// TIA Portal project "PLC_SecreTrap_V16" (V16)

(* hardware
DEVICE "S7-1200 station_1"  S7-1200 Station
   slot 0: "Rack_0"  S7-1200 Rack  Rack  V1.0
   slot 1: "PLC_1"  CPU 1212C DC/DC/DC  6ES7 212-1AE40-0XB0  V4.4
   slot 2: "DI 16/DQ 16x24VDC_1"  6ES7 223-1BL32-0XB0  V2.0
   slot 101: "CM 1241 (RS232)_1"  6ES7 241-1AH32-0XB0  V2.2
   slot 102: "CM 1241 (RS232)_2"  6ES7 241-1AH32-0XB0  V2.2
DEVICE "GSD device_1"  GSD.Device.PN
   slot 0: "Rack"  Rack  V1.0
   slot 0: "SINAMICS-S110-CU305PN-V4.4HF"  SINAMICS S110 CU305 PN V4.4HF/SP3  6SL3 040-0JA01-0AA0  V4.40
      slot 0: "SINAMICS S110 CU305 PN V4.4HF/SP3"  SINAMICS S110 CU305 PN V4.4HF/SP3
      slot 1: "PN-IO"  PN-IO
         slot 1: "Port 1"  Port 1
         slot 2: "Port 2"  Port 2
   slot 1: "DO Servo_1"  DO Servo
      slot 0: "Module Access Point:"  Module Access Point:
   slot 2: "DO Control Unit_1"  DO Control Unit
      slot 0: "Module Access Point:"  Module Access Point:
      slot 1: "without PROFIsafe"  without PROFIsafe
   slot 2: "Standard telegram 9, PZD-10/5"  Standard telegram 9, PZD-10/5
*)

// ===== PLC "PLC_1"  CPU 1212C DC/DC/DC =====

VAR_GLOBAL   // PLC tag table "Default tag table"
   "KM_Generator1" AT %Q0.0 : Bool;   // Contactor Generator 1
   "K_FunOFF_Generator1" AT %Q0.1 : Bool;   // Relay switch OFF Fun Generator 1
   "Tag_1" AT %M1.0 : Bool;
   "Tag_2" AT %M1.1 : Bool;
   "Tag_3" AT %M1.2 : Bool;
   "ONE" AT %M0.2 : Bool;
   "CycleInterrupt_Flag" AT %M10.0 : Bool;
   "KM_Generator2" AT %Q0.2 : Bool;   // Contactor Generator 2
   "K_FunOFF_Generator2" AT %Q0.3 : Bool;   // Relay switch OFF Fun Generator 2
   "Shutter2_LimPos1" AT %I0.5 : Bool;   // Limit switch Position 1 of Shutter 2
   "Shutter2_LimPos2" AT %I0.6 : Bool;   // Limit switch Position 2 of Shutter 2
   "Reserve1_IO" AT %I0.7 : Bool;   // Reserve 1
   "Clock_Byte" AT %MB100 : Byte;
   "Clock_10Hz" AT %M100.0 : Bool;
   "Clock_5Hz" AT %M100.1 : Bool;
   "Clock_2.5Hz" AT %M100.2 : Bool;
   "Clock_2Hz" AT %M100.3 : Bool;
   "Clock_1.25Hz" AT %M100.4 : Bool;
   "Clock_1Hz" AT %M100.5 : Bool;
   "Clock_0.625Hz" AT %M100.6 : Bool;
   "Clock_0.5Hz" AT %M100.7 : Bool;
   "Tag_4" AT %M1.3 : Bool;
   "Tag_5" AT %M1.4 : Bool;
   "Tag_6" AT %M1.5 : Bool;
   "Tag_7" AT %M1.6 : Bool;
   "EMG" AT %I0.2 : Bool;   // Emergency Stop key
   "Shutter1_LimPos1" AT %I0.3 : Bool;   // Limit switch Position 1 of Shutter 1
   "Resset_M" AT %M1.7 : Bool;
   "First_Scan" AT %M0.0 : Bool;
   "ZERO" AT %M0.3 : Bool;
   "DiagnosticStageChange" AT %M0.1 : Bool;
   "IR2" AT %I0.1 : Bool;   // Infrared sensor 2
   "IR1" AT %I0.0 : Bool;   // Infrared sensor 1
   "Shutter1_LimPos2" AT %I0.4 : Bool;   // Limit switch Position 2 of Shutter 1
   "OpenDoor_Key" AT %I1.0 : Bool;   // Open Door Key
   "CloseDoor_Key" AT %I1.1 : Bool;   // Close Door Key
   "QF_KM_Generator1" AT %I1.2 : Bool;   // State Contactor & Cercuit Breaker Generator 1
   "XRAY_Generator1" AT %I1.3 : Bool;   // X-RAY Status Generator 1
   "QF_KM_Generator2" AT %I1.4 : Bool;   // State Contactor & Cercuit Breaker Generator 2
   "XRAY_Generator2" AT %I1.5 : Bool;   // X-RAY Status Generator 2
   "RDY_Detectors" AT %I1.6 : Bool;   // Detectors is Ready to exposure
   "Fun1_Door" AT %I1.7 : Bool;   // State FUN 1 in the Door
   "Fun2_Door" AT %I2.0 : Bool;   // State FUN 2 in the Door
   "isLock_Door" AT %I2.1 : Bool;   // State Lock Door
   "Reserve2_IO" AT %I2.3 : Bool;   // Reserve 2
   "isClose_Door" AT %I2.4 : Bool;   // State Close Door
   "isFault_Door" AT %I2.5 : Bool;   // Active Fault Drive Door
   "Reserve3_IO" AT %I2.6 : Bool;   // Reserve 3
   "QF_KM_Door" AT %I2.7 : Bool;   // State QF for Door Power Source
   "QF_KM_Detectors" AT %I2.2 : Bool;   // State QF for Detector Power Source
   "K_Interlock_Generators" AT %Q0.4 : Bool;   // Relay Interlock Generators
   "Reserve1_DO" AT %Q0.6 : Bool;   // Reserve1 DO
   "Reserve2_DO" AT %Q0.7 : Bool;   // Reserve2 DO
   "K_Lock_Door" AT %Q1.0 : Bool;   // Relay Lock Door
   "HL_Door_Close" AT %Q1.1 : Bool;   // HL Door is Close
   "HL_XRAY_ON" AT %Q1.2 : Bool;   // HL X-RAY ON Status
   "TRIG_Detectors" AT %Q1.3 : Bool;   // TRIGGER to Detectors for Exposure
   "K_Fun1_Door" AT %Q1.4 : Bool;   // Relay switch ON Fun 1 Door
   "K_Fun2_Door" AT %Q1.5 : Bool;   // Relay switch ON Fun 2 Door
   "KM_Drive_Door" AT %Q1.6 : Bool;   // Contactor Drive Door
   "Reserve3_DO" AT %Q1.7 : Bool;   // Reserve 3 DO
   "Reserve4" AT %Q2.0 : Bool;   // Reserve 4 DO
   "HL_EMG" AT %Q2.1 : Bool;   // HL Emergency Stop
   "K_Open_Door" AT %Q2.3 : Bool;   // Relay Open Door
   "Reserve6_DO" AT %Q2.4 : Bool;   // Reserve6 DO
   "Reserve7_DO" AT %Q2.5 : Bool;   // Reserve7 DO
   "Reserve8_DO" AT %Q2.6 : Bool;   // Reserve8 DO
   "KM_Detectors" AT %Q2.2 : Bool;   // Contactor Detectors
   "K_Reserve" AT %Q2.7 : Bool;   // Relay Reserve
   "Tag_8" AT %Q0.5 : Bool;
END_VAR

VAR_GLOBAL CONSTANT   // PLC tag table "Default tag table"
   "LOW" : UInt := 1;
   "MIDLE" : UInt := 2;
   "HIGH" : UInt := 3;
   "NO_POWER" : UInt := 0;
   "STATUS_msg_Respose_timeout" : Word := 16#0097;   // The end of a message is recognized when there is no reply within a set time after transferring data
   "STATUS_RESPONSE_LENGHT" : Word := 16#0099;
   "STATUS_msg_CHAR_timeout" : Word := 16#0096;
   "STATUS_RESET_END" : Word := 16#0103;   // Reset complited
   "SUB_STATUS_NO_ERROR" : Word := 16#0000;
   "SYSTEM" : String := 'SYS0';   // device SYSTEM
   "GENERATOR1" : String := 'GEN1';
   "GENERATOR2" : String := 'GEN2';
   "STX" : Char := '2';
   "CR" : Char := 'D';
   "hash" : Char := '#';
   "addrSYS" : UInt := 1;   // device - System
   "addrGen1" : UInt := 2;   // device - Generator 1
   "addrGen2" : UInt := 3;   // device - Generator 2
   "addrShutter1" : UInt := 4;   // device - Shutter 1
   "addrShutter2" : UInt := 5;   // device - Shutter 2
   "addrDoor" : UInt := 6;   // device - Door
   "addrDetector" : UInt := 7;   // device - Detector
   "cmdSLEV" : UInt := 1;   // command Set Level (Presset)
   "cmdSCUR" : UInt := 3;   // command Set Current Generator
   "cmdSVLT" : UInt := 4;   // command Set Voltage Generator
   "cmdGCUR" : UInt := 5;   // command Get Current Generator
   "cmdGVLT" : UInt := 6;   // command Get Voltage Generator
   "SHUTTER1" : String := 'SHT1';
   "SHUTTER2" : String := 'SHT2';
   "DOOR" : String := 'DOOR';
   "DETECTOR" : String := 'DETC';
   "SETLEVEL" : String := 'SLEV';
   "GETLEVEL" : String := 'GLEV';
   "SETCURRENT" : String := 'SCUR';
   "SETVOLTAGE" : String := 'SVLT';
   "GETCURRENT" : String := 'GCUR';
   "GETVOLTAGE" : String := 'GVLT';
   "addrNOT" : UInt := 0;   // NOT device
   "cmdNOT" : UInt := 0;   // NOT command
   "STATUS_PC_REQ_ERROR" : Word := 16#0064;   // Error Request from PC
   "STATUS_PC_REQ_VAL_ERROR" : Word := 16#0065;   // Error Request from PC, Over value
   "cmdGLEV" : UInt := 2;   // command Get Level (Presset)
   "SETMODE" : String := 'SMOD';
   "GETMODE" : String := 'GMOD';
   "cmdSMOD" : UInt := 7;   // command Set Mode Scaner
   "cmdGMOD" : UInt := 8;   // command Get Mode Scaner
   "VP_max" : Real := 200.0;   // kV
   "VP_min" : Real := 80.0;   // kV
   "CP_max" : UInt := 6000;   // uA
   "CP_min" : UInt := 200;   // uA
   "Velo_max" : UInt := 45000;   // mm/min -> 145 ms
   "Velo_min" : UInt := 8450;   // mm/min -> 800 ms
   "SETWARM" : String := 'SWAR';
   "GETWARM" : String := 'GWAR';
   "cmdSWAR" : UInt := 9;   // command Set Warm UP Generator
   "cmdGWAR" : UInt := 10;   // command Get Warm UP Generator
   "FB_STATE_NO_PROCESSING" : UInt := 0;   // FB state: No processing
   "FB_STATE_VOLTAGE_PROGRAMM" : UInt := 1;   // FB state: Set Voltage
   "FB_STATE_CURRENT_PROGRAMM" : UInt := 2;   // FB state: Set Current
   "FB_STATE_MONITOR" : UInt := 3;   // FB state: Monitor
   "FB_STATE_FAULT_CLEAR" : UInt := 4;   // FB state: Fault Clear
   "FB_STATE_REPORT_FAULT" : UInt := 5;   // FB state: Report Fault
   "FB_STATE_HV_STATUS" : UInt := 6;   // FB state: HV Status
   "FB_STATE_X_RAY_ENABLE" : UInt := 7;   // FB state: X-RAY Enable
   "FB_STATE_WD_TIMER" : UInt := 8;   // FB state: Wath DOG Timer
   "FB_STATE_COMM_PORT_ECHO" : UInt := 9;   // FB state: Comm Port Echo
   "FB_STATE_WD_ENABLE" : UInt := 10;   // FB state: Watch Dog Enable/Disable
   "FB_STATE_WD_STATUS" : UInt := 11;   // FB state: Watch Dog
   "SETXRAY" : String := 'SRAY';
   "GETXRAY" : String := 'GRAY';
   "cmdSRAY" : UInt := 12;   // command Set X-RAY
   "cmdGRAY" : UInt := 11;   // command Get X-RAY
   "STATUS_msg_timeout" : UInt := 16#0095;
   "SETCLEAR" : String := 'SCLR';
   "cmdSCLR" : UInt := 13;   // command Reset
   "cmdGFLT" : UInt := 14;   // Command Get Fault
   "GETFAULT" : String := 'GFLT';
   "stageCycleShutter" : UInt := 10;   // Cycle Test Shutter
   "stageWaitGuest" : UInt := 0;   // Stage of waiting Guest
   "stagePrepareScan" : UInt := 1;   // Stage of preparing to scan
   "stageScaning" : UInt := 2;   // Stage of Scaning
   "stageOpenDoor" : UInt := 3;   // Stage of Opening the door
   "DRIVE1" : String := 'DRV1';   // device - Drive 1
   "DRIVE2" : String := 'DRV2';   // device - Drive 2
   "SETPOSITION" : String := 'SPOS';   // Set position of shutter
   "addrServoDrive1" : UInt := 8;   // device - Drive 1
   "addrServoDrive2" : UInt := 9;   // device - Drive 2
   "cmdSPOS" : UInt := 15;   // command positioning Drive
   "modeAUTO" : UInt := 3;   // mode AUTO
   "modeJOG" : UInt := 2;   // mode JOG
   "modeLIMITED" : UInt := 1;   // mode LIMITED
   "modeOFF" : UInt := 0;   // mode OFF
   "modeSERVIСE" : UInt := 4;   // mode Service
   "CountERR" : UInt := 3;   // Error Count
   "STATUS_SUBSEQUENT_CALL" : Word := 16#0102;   // Subsequent call during active processing without further details
   "STATUS_FIRST_CALL" : Word := 16#0101;   // First call after incoming new job (rising edge 'enable')
   "STATUS_NO_CALL" : Word := 16#0100;   // No job being currently processed
   "ERR_UNDEFINED_STATE" : Word := 16#0106;   // Error: due to an undefined state in state machine
   "ERR_Response_Generator" : Word := 16#0105;   // Error: response from generator not match argument CMD
   "ERR_NO_Response_Generator" : Word := 16#0104;   // Error: response from generator not match argument CMD
   "SETRESET" : String := 'SRES';
   "cmdSRES" : UInt := 16;   // command Set Reset logics
   "SETSCAN" : String := 'SCAN';   // Set Scan
   "cmdSCAN" : UInt := 17;   // command Set Scan
   "Xexposure" : DInt := 113000;   // Distance of shuter moove
   "AccShutter" : DInt := 57600;   // mm/min2, acceleration of shutter
   "TexposureMAX" : UInt := 800;   // ms, Maximum exposure time
   "TexposureMIN" : UInt := 145;   // ms, Minimum exposure time
   "SETPRES1" : String := 'SPR1';   // Set preset 1. Exposure tim in ms
   "SETPRES2" : String := 'SPR2';   // Set preset 2. Exposure tim in ms
   "SETPRES3" : String := 'SPR3';   // Set preset 3. Exposure tim in ms
   "cmdSPRESET1" : UInt := 18;   // Set preset 1. Exposure tim in ms
   "cmdSPRESET2" : UInt := 19;   // Set preset 2. Exposure tim in ms
   "cmdSPRESET3" : UInt := 20;   // Set preset 3. Exposure tim in ms
END_VAR

TYPE "typeGeneratorDATA"
   STRUCT
      VP_Programm : Real;   // Voltage Program
      CP_Programm : UInt;   // Current Program
      VP_Monitor : Real;   // Voltage Monitor
      CP_Monitor : UInt;   // Current Monitor
      T_Monitor : Real;   // Temperature Monitor
      FIL_Monitor : UInt;   // Filament Monitor
      X_RAY_Enable : Bool;   // Enable X-RAY
      X_RAY_Status : Bool;   // Monitir X-RAY status
      WDTE : Bool;   // Watch Dog Timer
      FREV : Bool;   // Comm Port Echo
      WDOG : Bool;   // Watch Dog Timer Enable/Disable
      WDOG_Status : Bool;
      FLT : Array[0..9] of Bool;   // Report Fault
      CMD_VP : Bool;   // Command Voltage Program
      CMD_CP : Bool;   // Command Current Program
      CMD_MON : Bool;   // Command Voltage/Current/Temperature/Filament Monitor
      CMD_CLR : Bool;   // Command Fault Clear
      CMD_FLT : Bool;   // Command Report Fault
      CMD_STAT : Bool;   // Command HV Status
      CMD_ENBL : Bool;   // Command X-Ray Enable
      CMD_WDTE : Bool;   // Command Watch Dog Timer
      CMD_FREV : Bool;   // Command Comm Port Echo
      CMD_WDOG : Bool;   // Command Watch Dog Enable/Disable
      CMD_WSTAT : Bool;   // Command Watch Dog Status
      CMD_CYCLE : Bool;   // CYCLE of executing Command
      CMD_VP_Ok : Bool;
      CMD_CP_Ok : Bool;
      DiagnosticCMD : Array[0..15] of "typeDiagnostics";
      cmd_Nunmber : UInt;   // Number executed command
      cmdDone : Bool;   // Command is done
      cmdError : Bool;   // Error
      cmdState : Word;   // Command status
   END_STRUCT;
   // // FLT[0] : Regulation
   // // FLT[1] : Interlock Open
   // // FLT[2] : Cathode Over KV Fault
   // // FLT[3] : Anode Over KV Fault
   // // FLT[4] : Over Temperature Fault
   // // FLT[5] : Arc Fault
   // // FLT[6] : Over Current Fault
   // // FLT[7] : Power Limit Fault
   // // FLT[8] : Over Voltage Fault
END_TYPE

TYPE "typeDiagnostics"
TITLE = typeDiagnosticsTemplate
   STRUCT
      status : Word;   // Status of the Block or error identification when error occurred
      count : UInt;   // Count of error occurred
   END_STRUCT;
END_TYPE

TYPE "typePresset"
   STRUCT
      VP : Real;   // Voltage rogramm
      CP : UInt;   // Current rogramm
      Velocity : DInt;   // Velocity shutter
      Texposure : UInt;   // Exposure time for shutter
      Ttrigger : Time;   // Trigger time for CareRay
   END_STRUCT;
END_TYPE

TYPE "typeTEL9"
   STRUCT
      OFF1 : Bool;   // 1 = On, 0 = Off (OFF1)
      OFF2 : Bool;   // 1 = No Coast Stop, 0 = Coast Stop (OFF2)
      OFF3 : Bool;   // 1 = No Quick Stop, 0 = Quick Stop (OFF3)
      enableOperation : Bool;   // 1 = Enable operation
      rejectTraversingTask : Bool;   // 0 = Reject active traversing task
      intermediateStop : Bool;   // 0 = Intermediate STOP active traversing task
      acknowledgeError : Bool;   // Acknowledge faults (0 -> 1)
      jog1 : Bool;   // Jog 1 signal
      jog2 : Bool;   // Jog 2 signal
      startHomingProcedure : Bool;   // Start homing procedure
      activateTraversingTask : Bool;   // Activate traversing task
      traversingTaskSelection : UInt;   // Select traversing task (0..1023)
      submode : Bool;   // Submode: 0 = program 1 = Manual data input (MDI)
      stw2 : Word;   // Control word 2 (STW2)
      targetPositionMDI : DInt;   // MDI target position
      velocityMDI : DInt;   // MDI velocity
      accelerationOverrideMDI : Real;   // MDI override of acceleration [%]
      decelerationOverrideMDI : Real;   // MDI override of deceleration [%]
      positioningModeMDI : Bool;   // Positioning 0 = relative 1 = absolute
      directionPositiveMDI : Bool;   // Modulo axis: Absolute positioning in positive direction. If directionPosMDI = directionNegMDI positioning via shortest way.
      directionNegativeMDI : Bool;   // Modulo axis: Absolute positioning in negative direction. If directionNegMDI = directionPosMDI positioning via shortest way.
      operationEnabled : Bool;   // Operation enabled
      switchingOnInhibited : Bool;   // Switching on inhibited
      faultActive : Bool;   // Fault present
      warningActive : Bool;   // Warning present
      homePositionSet : Bool;   // Home position set (axis homed)
      targetPositionReached : Bool;   // Target position reached
      driveStopped : Bool;   // A traversing task has been completed or standstill for intermediate stop
      traversingTaskAcknowledged : Bool;   // A new traversing task or MDI setpoint was started
      actualPosition : DInt;   // Actual position
      activeTraversingTask : UInt;   // Active traversing task
      zsw1 : Word;   // Status word 1
      zsw2 : Word;   // Status word 2
      error : Bool;   // Error active, check status and diagId
      status : Word;   // Status output (7002 = FB in operation; 8xxx = error code)
      diagId : DWord;   // Error codes of the cyclic system function blocks GETIO / SETIO
   END_STRUCT;
END_TYPE

TYPE "typeREQ"
   STRUCT
      STX : Byte := '2';
      ADDR : Array[0..3] of Byte;
      hash1 : Byte := '#';
      CMD : Array[0..3] of Byte;
      hash2 : Byte := '#';
      VALUE : Array[0..3] of Byte;
      CR : Byte := 'D';
   END_STRUCT;
END_TYPE

TYPE "typeRESP"
   STRUCT
      STX : Byte := '2';
      ADDR : Array[0..3] of Byte;
      hash1 : Byte := '#';
      CMD : Array[0..3] of Byte;
      hash2 : Byte := '#';
      VALUE : Array[0..3] of Byte;
      CR : Byte := 'D';
   END_STRUCT;
END_TYPE

TYPE "typeWarmTable"
   STRUCT
      VP : Array[1..10] of Real;
      CP : Array[1..10] of UInt;
      T : Array[1..3] of Time;
   END_STRUCT;
END_TYPE

DATA_BLOCK "temp"   // DB2
{ S7_Optimized_Access := 'TRUE' }
VERSION : 0.1
   VAR RETAIN
      Time_Temp : Array[0..18] of DTL;
      Temperature : Array[0..18] of Real;
      index_temperature : UInt;
   END_VAR
   VAR
      "test.temperature_EN" : Bool;
      temp_XRAY_ON : Bool;
      front : Bool;
      rise1 : Bool;
      rize2 : Bool;
      cycleShutter : Bool;
      "T1_X-RAY" : DTL;
      "T2_X-RAY" : DTL;
      T_XRAY : Time;
      rise2 : Bool;
      para : UInt;
      err : Bool;
   END_VAR
BEGIN
END_DATA_BLOCK

// folder: CMD

DATA_BLOCK "PCtoPLC_DB"   // DB12
{ S7_Optimized_Access := 'TRUE' }
VERSION : 0.1
// stored: InstanceOfName ParcingCMD
"ParcingCMD"
BEGIN
END_DATA_BLOCK

DATA_BLOCK "SateMaсhineCMD_DB"   // DB15
{ S7_Optimized_Access := 'TRUE' }
VERSION : 0.1
// stored: InstanceOfName SateMaсhineCMD
"SateMaсhineCMD"
BEGIN
END_DATA_BLOCK

// folder: Drive

DATA_BLOCK "DriveStage_DB_1"   // DB7
{ S7_Optimized_Access := 'TRUE' }
VERSION : 0.1
// stored: InstanceOfName DrivesStage
"DrivesStage"
BEGIN
END_DATA_BLOCK

DATA_BLOCK "PD_TEL9_DrivePos_DB_1"   // DB17
{ S7_Optimized_Access := 'TRUE' }
AUTHOR : SIEMENS
VERSION : 0.1
// stored: InstanceOfName PD_TEL9_DrivePos
"PD_TEL9_DrivePos"
BEGIN
END_DATA_BLOCK

DATA_BLOCK "TEL9_Drive1"   // DB20
{ S7_Optimized_Access := 'TRUE' }
VERSION : 0.1
BEGIN
END_DATA_BLOCK

DATA_BLOCK "DriveStage_DB_2"   // DB41
{ S7_Optimized_Access := 'TRUE' }
VERSION : 0.1
// stored: InstanceOfName DrivesStage
"DrivesStage"
BEGIN
END_DATA_BLOCK

DATA_BLOCK "PD_TEL9_DrivePos_DB_2"   // DB42
{ S7_Optimized_Access := 'TRUE' }
AUTHOR : SIEMENS
VERSION : 0.1
// stored: InstanceOfName PD_TEL9_DrivePos
"PD_TEL9_DrivePos"
BEGIN
END_DATA_BLOCK

DATA_BLOCK "TEL9_Drive2"   // DB43
{ S7_Optimized_Access := 'TRUE' }
VERSION : 0.1
BEGIN
END_DATA_BLOCK

// folder: Generators

DATA_BLOCK "Generator1_DIO_DB"   // DB1
{ S7_Optimized_Access := 'TRUE' }
VERSION : 0.1
// stored: InstanceOfName GeneratorDIO
"GeneratorDIO"
BEGIN
   statString := '7770';
END_DATA_BLOCK

DATA_BLOCK "WarmTable"   // DB3
{ S7_Optimized_Access := 'TRUE' }
VERSION : 0.1
BEGIN
   T[1] := T#300s;
   T[2] := T#60s;
   T[3] := T#30s;
   VP[1] := 80.0;
   VP[2] := 90.0;
   VP[3] := 100.0;
   VP[4] := 110.0;
   VP[5] := 120.0;
   VP[6] := 130.0;
   VP[7] := 140.0;
   VP[8] := 150.0;
   VP[9] := 160.0;
   VP[10] := 160.0;
   CP[1] := 200;
   CP[2] := 530;
   CP[3] := 860;
   CP[4] := 1190;
   CP[5] := 1520;
   CP[6] := 1850;
   CP[7] := 2180;
   CP[8] := 2510;
   CP[9] := 2840;
   CP[10] := 3120;
END_DATA_BLOCK

DATA_BLOCK "GeneratorDATA_1"   // DB6
{ S7_Optimized_Access := 'TRUE' }
VERSION : 0.1
BEGIN
END_DATA_BLOCK

DATA_BLOCK "GenOperate1_DB"   // DB8
{ S7_Optimized_Access := 'TRUE' }
VERSION : 0.1
// stored: InstanceOfName GenOperate
"GenOperate"
BEGIN
END_DATA_BLOCK

DATA_BLOCK "GenOperate2_DB"   // DB16
{ S7_Optimized_Access := 'TRUE' }
VERSION : 0.1
// stored: InstanceOfName GenOperate
"GenOperate"
BEGIN
END_DATA_BLOCK

DATA_BLOCK "GeneratorWarm1_DB"   // DB34
{ S7_Optimized_Access := 'TRUE' }
VERSION : 0.1
// stored: InstanceOfName GeneratorWarm
"GeneratorWarm"
BEGIN
END_DATA_BLOCK

DATA_BLOCK "GeneratorDATA_2"   // DB36
{ S7_Optimized_Access := 'TRUE' }
VERSION : 0.1
BEGIN
END_DATA_BLOCK

DATA_BLOCK "GeneratorWarm2_DB"   // DB51
{ S7_Optimized_Access := 'TRUE' }
VERSION : 0.1
// stored: InstanceOfName GeneratorWarm
"GeneratorWarm"
BEGIN
END_DATA_BLOCK

DATA_BLOCK "Generator2_DIO_DB"   // DB52
{ S7_Optimized_Access := 'TRUE' }
VERSION : 0.1
// stored: InstanceOfName GeneratorDIO
"GeneratorDIO"
BEGIN
   statString := '7770';
END_DATA_BLOCK

// folder: Global_DATA

DATA_BLOCK "DIODATA"   // DB9
{ S7_Optimized_Access := 'TRUE' }
VERSION : 0.1
   VAR
      DI : Struct
         IR1_I0_0 : Bool;   // Infrared Sensor 1
         IR2_I0_1 : Bool;   // Infrared Sensor 2
         EMG_I0_2 : Bool;   // Key Emergensy Stop
         Pos1_Shutter1_I0_3 : Bool;   // Position Switch 1 of Shutter 1
         Pos2_Shutter1_I0_4 : Bool;   // Position Switch 2 of Shutter 1
         Pos1_Shutter2_I0_5 : Bool;   // Position Switch 2 of Shutter 1
         Pos2_Shutter2_I0_6 : Bool;   // Position Switch 2 of Shutter 1
         Reserve1_I0_7 : Bool;   // Reserve1
         OpenDoor_I1_0 : Bool;   // Key Open Door
         CloseDoor_I1_1 : Bool;   // Key Close Door
         QF_KM_Drive1_I1_2 : Bool;   // State Contactor & Cercuit Breaker Drive 1
         XRAY_Generator1_I1_3 : Bool;   // X-RAY Status Generator 1
         QF_KM_Drive2_I1_4 : Bool;   // State Contactor & Cercuit Breaker Drive 2
         XRAY_Generator2_I1_5 : Bool;   // X-RAY Status Generator 2
         RDY_Detectors_I1_6 : Bool;   // Detectors is Ready to exposure
         Fun1_Door_I1_7 : Bool;   // State FUN 1 in the Door
         Fun2_Door_I2_0 : Bool;   // State FUN 2 in the Door
         LockDoor_I2_1 : Bool;   // State Lock Door
         QF_KM_Detectors_I2_2 : Bool;   // State QF for Detector Power Source
         Reserve2_I2_3 : Bool;   // Reserve2
         Close_Door_I2_4 : Bool;   // State Close Door
         Fault_Door_I2_5 : Bool;   // State Fault Drive Door
         Reserve3_I2_6 : Bool;   // Reserve3
         Reserve4_I2_7 : Bool;   // Reserve4
      END_STRUCT;
      "DO" : Struct
         KM_Drive1_Q0_0 : Bool;   // Contactor Drive 1
         K_FunOFF_Generator1_Q0_1 : Bool;   // Relay switch OFF Fun Generator 1
         KM_Drive2_Q0_2 : Bool;   // Contactor Drive 2
         K_FunOFF_Generator2_Q0_3 : Bool;   // Relay switch OFF Fun Generator 2
         K_Interlock_Generators_Q0_4 : Bool;   // Relay Interlock Generators
         K_Open_Door_Q0_5 : Bool;   // Relay Open Door
         Reserve1_Q0_6 : Bool;   // Reserve 1 DO
         Reserve2_Q0_7 : Bool;   // Reserve 2 DO
         K_Lock_Door_Q1_0 : Bool;   // Relay Lock Door
         HL_Door_Close_Q1_1 : Bool;   // HL Door is Close
         HL_XRAY_ON_Q1_2 : Bool;   // HL X-RAY ON Status
         TRIG_Detectors_Q1_3 : Bool;   // TRIGGER to Detectors for Exposure
         K_Fun1_Door_Q1_4 : Bool;   // Relay switch ON Fun 1 Door
         K_Fun2_Door_Q1_5 : Bool;   // Relay switch ON Fun 2 Door
         KM_Drive_Door_Q1_6 : Bool;   // Contactor Drive Door
         Reserve3_Q1_7 : Bool;   // Reserve 3 DO
         Reserve4_Q2_0 : Bool;   // Reserve 4 DO
         HL_EMG_Q2_1 : Bool;   // HL Emergency Stop
         KM_Detectors_Q2_2 : Bool;   // Contactor Detectors
         Reserve5_Q2_3 : Bool;   // Reserve 5 DO
         Reserve6_Q2_4 : Bool;   // Reserve 6 DO
         Reserve7_Q2_5 : Bool;   // Reserve 7 DO
         Reserve8_Q2_6 : Bool;   // Reserve 8 DO
         K_Reserve_Q2_7 : Bool;   // Relay Reserve
      END_STRUCT;
   END_VAR
BEGIN
END_DATA_BLOCK

DATA_BLOCK "CmdDATA"   // DB10
{ S7_Optimized_Access := 'TRUE' }
VERSION : 0.1
   VAR
      REQ : String[16] := '               ';
      RESP : String[16] := '               ';
   END_VAR
BEGIN
END_DATA_BLOCK

DATA_BLOCK "PressetDATA"   // DB13
{ S7_Optimized_Access := 'TRUE' }
VERSION : 0.1
   VAR RETAIN
      Shutter1 : Struct
         POS1 : DInt := 5000;   // um Position Start Sgutter
         POS2 : DInt := 147000;   // um Position Stop Sgutter
      END_STRUCT;
      Shutter2 : Struct
         POS1 : DInt := 5000;   // um Position Start Sgutter
         POS2 : DInt := 147000;   // um Position Stop Sgutter
      END_STRUCT;
      GUEST : Array[0..3] of "typePresset";
   END_VAR
BEGIN
   GUEST[0].Velocity := 0;   // mm/min
   GUEST[1].Velocity := 8480;   // 8480 mm/min 800 ms
   GUEST[2].Velocity := 17000;   // 17000 mm/min 400 ms
   GUEST[3].Velocity := 45000;   // 45000 mm/min 145 ms
   GUEST[1].VP := 80.0;   // kV
   GUEST[1].CP := 200;   // uA
   GUEST[2].VP := 80.0;   // kV
   GUEST[2].CP := 200;   // uA
   GUEST[3].VP := 80.0;   // kV
   GUEST[3].CP := 200;   // uA
   GUEST[1].Texposure := 800;
   GUEST[2].Texposure := 400;
   GUEST[3].Texposure := 140;
   // GUEST[0].VP : kV
   // GUEST[0].CP : uA
END_DATA_BLOCK

DATA_BLOCK "GlobalDATA"   // DB14
{ S7_Optimized_Access := 'TRUE' }
VERSION : 0.1
   VAR
      N_Presset : UInt := 0;   // 0 - NO Scan, 1 - Low. 2 - Medium, 3 - High
      CountShot : UInt := 2;   // 1- one shot, 2- two shot
      modeDrive : Bool;   // 0-MDI 1-JOG
      readyToScan : Bool;   // 0 - is not ready to scan, 1- ready to scan
      readyData : Bool;   // 0 - Images not ready, 1 - Images ready
      modeScan : UInt := 0;   // 0 to 4. 0 - OFF, 1 - Limited, 2-JOG, 3-AUTO, 4-Service
      stageScan : UInt;   // 0 - WaitGuest, 1 - PrepareScan, 2 - Scaning, 3 - OpenDoor
      startScan : Bool;   // 0 - no Scan, 1 - Set Scan
      newPreset : Bool;   // 0 - no Preset, 1- recive new preset
      Scan_XRAY : Bool;   // 0 - Scan without XRAY, 1 - Scan with X-RAY
      cmdReset : Struct   // Resset Command
         Global : Bool;   // Reset global logic
         Drive1 : Bool;   // Reset drive 1 logic and Fault
         Drive2 : Bool;   // Reset drive 2 logic and Fault
         Generator1 : Bool;   // Reset Generator 1 logic
         Generator2 : Bool;   // Reset Generator 2 logic
         Door : Bool;   // Reset Drive door
         Detector : Bool;   // Reset Detector logic
      END_STRUCT;
      Shutter1 : Struct   // Command and state of Shutter 1
         cmdCycle : Bool;   // Command cycle moving in Service mode
         cmdPOS1 : Bool;   // Command move shutter to Position 1
         cmdPOS2 : Bool;   // Command move shutter to Position 2
         cmdOFF1 : Bool;   // Command pulse enable Drive (ON/OFF1)
         Ready : Bool;   // Drive Ready/ 1 - ON, 0 - OFF
         Position : DInt;   // Current position (um)
         Velocity : DInt;   // Setpoint velocity
         setPOS1 : Bool;   // Сommand executed (Shutter in POS1)
         setPOS2 : Bool;   // Сommand executed (Shutter in POS2)
         faulActive : Bool;   // Drive has Fault
         powerFail : Bool;   // KM or QF of power drive is Fail
      END_STRUCT;
      Shutter2 : Struct   // Command and state of Shutter 2
         cmdCycle : Bool;   // Command cycle moving in Service mode
         cmdPOS1 : Bool;   // Command move shutter to Position 1
         cmdPOS2 : Bool;   // Command move shutter to Position 2
         cmdOFF1 : Bool;   // Command pulse enable Drive (ON/OFF1)
         Ready : Bool;   // Drive Ready/ 1 - ON, 0 - OFF
         Position : DInt;   // Current position (um)
         Velocity : DInt;   // Setpoint velocity
         setPOS1 : Bool;   // Сommand executed (Shutter in POS1)
         setPOS2 : Bool;   // Сommand executed (Shutter in POS2)
         faulActive : Bool;   // Drive has Fault
         powerFail : Bool;   // KM or QF of power drive is Fail
      END_STRUCT;
      Generator1 : Struct   // Command and state of Generator 1
         Enable : Bool := true;   // Enable generator to shot
         Ready : Bool;   // Ready to work
         cmdWarm : UInt;   // Warm Up. 0- NO warm, 1-Table1, 2-Table2, 3-Table3
         warmTimeOFF : Time;   // Time out of Warm
         warmEN : Bool;   // Warm enabled (curently executing)
         warmDone : Bool;   // Warming was done
         VP : Real;   // Voltage programm (kV)
         CP : UInt;   // Current programm (uA)
         VP_monitor : Real;   // Voltage monitoring (kV)
         CP_monitor : UInt;   // Current monitoring (uA)
         T_monitor : Real;   // Temperature monitoring (C)
         FLT : Array[0..9] of Bool;   // Fault
         CmdXRAY_ON : Bool;   // Command to X-RAY swith ON (1 - ON, 0 - OFF)
         XRAY_Status : Bool;   // Status of X-RAY (1- ON, 0 - OFF)
         PWR_Status : Bool;   // Power status of XRAY (VP=VP_monitor, CP=CP_monitor)
         Fault : Bool;   // Fault of RS232 interface (0 - NO Fault, 1 - Fault active))
         PowerFail : Bool;   // KM or QF of power drive is Fail
         RS232_Status : Word;   // Status of RS232 interface (status word)
      END_STRUCT;
      Generator2 : Struct   // Command and state of Generator 2
         Enable : Bool;   // Enable generator to shot
         Ready : Bool;   // Ready to work
         cmdWarm : UInt;   // Warm Up. 0- NO warm, 1-Table1, 2-Table2, 3-Table3
         warmTimeOFF : Time;   // Time out of Warm
         warmEN : Bool;   // Warm enabled (curently executing)
         warmDone : Bool;   // Warming was done
         VP : Real;   // Voltage programm (kV)
         CP : UInt;   // Current programm (uA)
         VP_monitor : Real;   // Voltage monitoring (kV)
         CP_monitor : UInt;   // Current monitoring (uA)
         T_monitor : Real;   // Temperature monitoring (C)
         FLT : Array[0..9] of Bool;   // Fault
         CmdXRAY_ON : Bool;   // Command to X-RAY swith ON (1 - ON, 0 - OFF)
         XRAY_Status : Bool;   // Status of X-RAY (1- ON, 0 - OFF)
         PWR_Status : Bool;   // Power status of XRAY (VP=VP_monitor, CP=CP_monitor)
         Fault : Bool;   // Fault of RS232 interface (0 - NO Fault, 1 - Fault active))
         PowerFail : Bool;   // KM or QF of power drive is Fail
         RS232_Status : Word;   // Status of RS232 interface (status word)
      END_STRUCT;
      Door : Struct   // Command and state of Door
         CmdOpen : Bool;   // Comman to open the DOOR (1 - open, 0 - close)
         CmdLock : Bool;   // Command to lock the DOOR (1 - lock, 0 - unlock)
         CmdReset : Bool;   // Command to resset drive (1 - resset, 0 - resset)
         cmdFan : Bool;   // Command to switch OFF Cooling Fans
         isClose : Bool;   // State of the DOOR (1 - close, 0 - open)
         isLock : Bool;   // State of the DOOR (1 - lock, 0 - unlock)
         faulActive : Bool;   // Fault Active of drive the door (1 - Faul Present, 0 - 1 - no Fault )
         PowerFail : Bool;   // KM or QF of power drive is Fail
         Temperature : Real;   // Temperature inside the door (C)
      END_STRUCT;
      Detector : Struct   // Command and state of Detector
         PowerFail : Bool;   // KM or QF of power drive is Fail
         MoxaFail : Bool;   // Switch MOXA has Fail
      END_STRUCT;
      REQ : Struct   // structure request
         ADDR : UInt;   // addres device
         CMD : UInt;   // Command
         Value : UInt;   // Value
         Error : Bool;   // Request has error
      END_STRUCT;
      RESP : Struct   // structure respoce
         ADDR : UInt;   // addres device
         CMD : UInt;   // Command
         Value : UInt;   // Value
         Done : Bool;   // Command complited
      END_STRUCT;
   END_VAR
BEGIN
   // Generator1.FLT[0] : 0 - No Regulation Fault, 1 - Regulation
   // Generator1.FLT[1] : 0 - No Interlock Open, 1 - Interlock Open
   // Generator1.FLT[2] : 0 - No Fault, 1 - Cathode Over KV Fault
   // Generator1.FLT[3] : 0 - No Fault, 1 - Anode Over KV Fault
   // Generator1.FLT[4] : 0 - No Fault, 1 - Over Temperature Fault
   // Generator1.FLT[5] : 0 - No Fault, 1 - Arc Fault
   // Generator1.FLT[6] : 0 - No Fault, 1 - Over Current Fault
   // Generator1.FLT[7] : 0 - No Fault, 1- Power Limit Fault
   // Generator1.FLT[8] : 0 - No Fault, 1 - Over Voltage Fault
   // Generator1.FLT[9] : 0 - No Fault,
   // Generator2.FLT[0] : 0 - No Regulation Fault, 1 - Regulation
   // Generator2.FLT[1] : 0 - No Interlock Open, 1 - Interlock Open
   // Generator2.FLT[2] : 0 - No Fault, 1 - Cathode Over KV Fault
   // Generator2.FLT[3] : 0 - No Fault, 1 - Anode Over KV Fault
   // Generator2.FLT[4] : 0 - No Fault, 1 - Over Temperature Fault
   // Generator2.FLT[5] : 0 - No Fault, 1 - Arc Fault
   // Generator2.FLT[6] : 0 - No Fault, 1 - Over Current Fault
   // Generator2.FLT[7] : 0 - No Fault, 1- Power Limit Fault
   // Generator2.FLT[8] : 0 - No Fault, 1 - Over Voltage Fault
   // Generator2.FLT[9] : 0 - No Fault,
END_DATA_BLOCK

// folder: IR

DATA_BLOCK "IR"   // DB11
{ S7_Optimized_Access := 'TRUE' }
VERSION : 0.1
   VAR
      Guest : Array[0..5] of Struct
         IR1 : Array[0..5] of Struct
            t1 : DTL;
            t2 : DTL;
            delta : Time;
         END_STRUCT;
         IR1_t1 : DTL;
         IR2_t1 : DTL;
         Delta_IR2_IR1 : Time;
         count : Int;
      END_STRUCT;
      Guest_came : Bool;
      Guest_index : Int;
      IR1_count : Int;
      IR1_t1 : DTL;
      IR1_t2 : DTL;
      IR2_t1 : DTL;
      Delta_IR2_IR1 : Time;
      SHOT_make : Bool;
   END_VAR
BEGIN
END_DATA_BLOCK

// folder: Safety

DATA_BLOCK "Safety_DB"   // DB31
{ S7_Optimized_Access := 'TRUE' }
VERSION : 0.1
// stored: InstanceOfName Safety
"Safety"
BEGIN
END_DATA_BLOCK

// folder: StatMachine

DATA_BLOCK "StatMachine_DB"   // DB25
{ S7_Optimized_Access := 'TRUE' }
VERSION : 0.1
// stored: InstanceOfName StatMachineGLOBAL
"StatMachineGLOBAL"
BEGIN
END_DATA_BLOCK

// folder: System blocks/Program resources

DATA_BLOCK "IEC_Timer_0_DB_11"   // DB23
{ S7_Optimized_Access := 'TRUE' }
AUTHOR : Simatic
FAMILY : IEC
NAME : IEC_TMR
VERSION : 1.0
// stored: InstanceOfName IEC_TIMER
"IEC_TIMER"
BEGIN
END_DATA_BLOCK

DATA_BLOCK "IEC_Timer_0_DB_2"   // DB24
{ S7_Optimized_Access := 'TRUE' }
AUTHOR : Simatic
FAMILY : IEC
NAME : IEC_TMR
VERSION : 1.0
// stored: InstanceOfName IEC_TIMER
"IEC_TIMER"
BEGIN
END_DATA_BLOCK

DATA_BLOCK "IEC_Timer_0_DB_3"   // DB26
{ S7_Optimized_Access := 'TRUE' }
AUTHOR : Simatic
FAMILY : IEC
NAME : IEC_TMR
VERSION : 1.0
// stored: InstanceOfName IEC_TIMER
"IEC_TIMER"
BEGIN
END_DATA_BLOCK

DATA_BLOCK "IEC_Timer_0_DB_4"   // DB27
{ S7_Optimized_Access := 'TRUE' }
AUTHOR : Simatic
FAMILY : IEC
NAME : IEC_TMR
VERSION : 1.0
// stored: InstanceOfName IEC_TIMER
"IEC_TIMER"
BEGIN
END_DATA_BLOCK

DATA_BLOCK "IEC_Timer_0_DB_5"   // DB28
{ S7_Optimized_Access := 'TRUE' }
AUTHOR : Simatic
FAMILY : IEC
NAME : IEC_TMR
VERSION : 1.0
// stored: InstanceOfName IEC_TIMER
"IEC_TIMER"
BEGIN
END_DATA_BLOCK

DATA_BLOCK "IEC_Timer_0_DB_6"   // DB29
{ S7_Optimized_Access := 'TRUE' }
AUTHOR : Simatic
FAMILY : IEC
NAME : IEC_TMR
VERSION : 1.0
// stored: InstanceOfName IEC_TIMER
"IEC_TIMER"
BEGIN
END_DATA_BLOCK

DATA_BLOCK "IEC_Timer_0_DB_7"   // DB30
{ S7_Optimized_Access := 'TRUE' }
AUTHOR : Simatic
FAMILY : IEC
NAME : IEC_TMR
VERSION : 1.0
// stored: InstanceOfName IEC_TIMER
"IEC_TIMER"
BEGIN
END_DATA_BLOCK

DATA_BLOCK "IEC_Timer_0_DB_8"   // DB32
{ S7_Optimized_Access := 'TRUE' }
AUTHOR : Simatic
FAMILY : IEC
NAME : IEC_TMR
VERSION : 1.0
// stored: InstanceOfName IEC_TIMER
"IEC_TIMER"
BEGIN
END_DATA_BLOCK

DATA_BLOCK "IEC_Timer_0_DB_10"   // DB33
{ S7_Optimized_Access := 'TRUE' }
AUTHOR : Simatic
FAMILY : IEC
NAME : IEC_TMR
VERSION : 1.0
// stored: InstanceOfName IEC_TIMER
"IEC_TIMER"
BEGIN
END_DATA_BLOCK

DATA_BLOCK "IEC_Timer_0_DB_9"   // DB35
{ S7_Optimized_Access := 'TRUE' }
AUTHOR : Simatic
FAMILY : IEC
NAME : IEC_TMR
VERSION : 1.0
// stored: InstanceOfName IEC_TIMER
"IEC_TIMER"
BEGIN
END_DATA_BLOCK

DATA_BLOCK "IEC_Timer_0_DB_12"   // DB37
{ S7_Optimized_Access := 'TRUE' }
AUTHOR : Simatic
FAMILY : IEC
NAME : IEC_TMR
VERSION : 1.0
// stored: InstanceOfName IEC_TIMER
"IEC_TIMER"
BEGIN
END_DATA_BLOCK

DATA_BLOCK "IEC_Timer_0_DB_13"   // DB38
{ S7_Optimized_Access := 'TRUE' }
AUTHOR : Simatic
FAMILY : IEC
NAME : IEC_TMR
VERSION : 1.0
// stored: InstanceOfName IEC_TIMER
"IEC_TIMER"
BEGIN
END_DATA_BLOCK

DATA_BLOCK "IEC_Timer_0_DB_14"   // DB39
{ S7_Optimized_Access := 'TRUE' }
AUTHOR : Simatic
FAMILY : IEC
NAME : IEC_TMR
VERSION : 1.0
// stored: InstanceOfName IEC_TIMER
"IEC_TIMER"
BEGIN
END_DATA_BLOCK

DATA_BLOCK "IEC_Timer_0_DB_15"   // DB40
{ S7_Optimized_Access := 'TRUE' }
AUTHOR : Simatic
FAMILY : IEC
NAME : IEC_TMR
VERSION : 1.0
// stored: InstanceOfName IEC_TIMER
"IEC_TIMER"
BEGIN
END_DATA_BLOCK

DATA_BLOCK "IEC_Timer_0_DB_16"   // DB44
{ S7_Optimized_Access := 'TRUE' }
AUTHOR : Simatic
FAMILY : IEC
NAME : IEC_TMR
VERSION : 1.0
// stored: InstanceOfName IEC_TIMER
"IEC_TIMER"
BEGIN
END_DATA_BLOCK

DATA_BLOCK "IEC_Timer_0_DB_17"   // DB45
{ S7_Optimized_Access := 'TRUE' }
AUTHOR : Simatic
FAMILY : IEC
NAME : IEC_TMR
VERSION : 1.0
// stored: InstanceOfName IEC_TIMER
"IEC_TIMER"
BEGIN
END_DATA_BLOCK

DATA_BLOCK "IEC_Timer_0_DB_18"   // DB46
{ S7_Optimized_Access := 'TRUE' }
AUTHOR : Simatic
FAMILY : IEC
NAME : IEC_TMR
VERSION : 1.0
// stored: InstanceOfName IEC_TIMER
"IEC_TIMER"
BEGIN
END_DATA_BLOCK

DATA_BLOCK "IEC_Timer_0_DB_19"   // DB47
{ S7_Optimized_Access := 'TRUE' }
AUTHOR : Simatic
FAMILY : IEC
NAME : IEC_TMR
VERSION : 1.0
// stored: InstanceOfName IEC_TIMER
"IEC_TIMER"
BEGIN
END_DATA_BLOCK

DATA_BLOCK "IEC_Timer_0_DB_20"   // DB48
{ S7_Optimized_Access := 'TRUE' }
AUTHOR : Simatic
FAMILY : IEC
NAME : IEC_TMR
VERSION : 1.0
// stored: InstanceOfName IEC_TIMER
"IEC_TIMER"
BEGIN
END_DATA_BLOCK

DATA_BLOCK "IEC_Timer_0_DB_21"   // DB49
{ S7_Optimized_Access := 'TRUE' }
AUTHOR : Simatic
FAMILY : IEC
NAME : IEC_TMR
VERSION : 1.0
// stored: InstanceOfName IEC_TIMER
"IEC_TIMER"
BEGIN
END_DATA_BLOCK

DATA_BLOCK "IEC_Timer_0_DB_22"   // DB50
{ S7_Optimized_Access := 'TRUE' }
AUTHOR : Simatic
FAMILY : IEC
NAME : IEC_TMR
VERSION : 1.0
// stored: InstanceOfName IEC_TIMER
"IEC_TIMER"
BEGIN
END_DATA_BLOCK

DATA_BLOCK "IEC_Timer_0_DB_23"   // DB53
{ S7_Optimized_Access := 'TRUE' }
AUTHOR : Simatic
FAMILY : IEC
NAME : IEC_TMR
VERSION : 1.0
// stored: InstanceOfName IEC_TIMER
"IEC_TIMER"
BEGIN
END_DATA_BLOCK

DATA_BLOCK "IEC_Timer_0_DB_24"   // DB54
{ S7_Optimized_Access := 'TRUE' }
AUTHOR : Simatic
FAMILY : IEC
NAME : IEC_TMR
VERSION : 1.0
// stored: InstanceOfName IEC_TIMER
"IEC_TIMER"
BEGIN
END_DATA_BLOCK

DATA_BLOCK "IEC_Timer_0_DB_25"   // DB55
{ S7_Optimized_Access := 'TRUE' }
AUTHOR : Simatic
FAMILY : IEC
NAME : IEC_TMR
VERSION : 1.0
// stored: InstanceOfName IEC_TIMER
"IEC_TIMER"
BEGIN
END_DATA_BLOCK

// folder: (top level)

ORGANIZATION_BLOCK "Main"   // OB1, LAD, ProgramCycle
TITLE = "Main Program Sweep (Cycle)"
{ S7_Optimized_Access := 'TRUE' }
VERSION : 0.1
   VAR_INPUT
      Initial_Call : Bool;   // Initial call of this OB
      Remanence : Bool;   // =True, if remanent data are available
   END_VAR
   VAR_TEMP
      temp1 : Bool;
      temp2 : Bool;
      temp3 : Bool;
      temp3_old : Bool;
   END_VAR
BEGIN

REGION Network 1: Блок безопасности
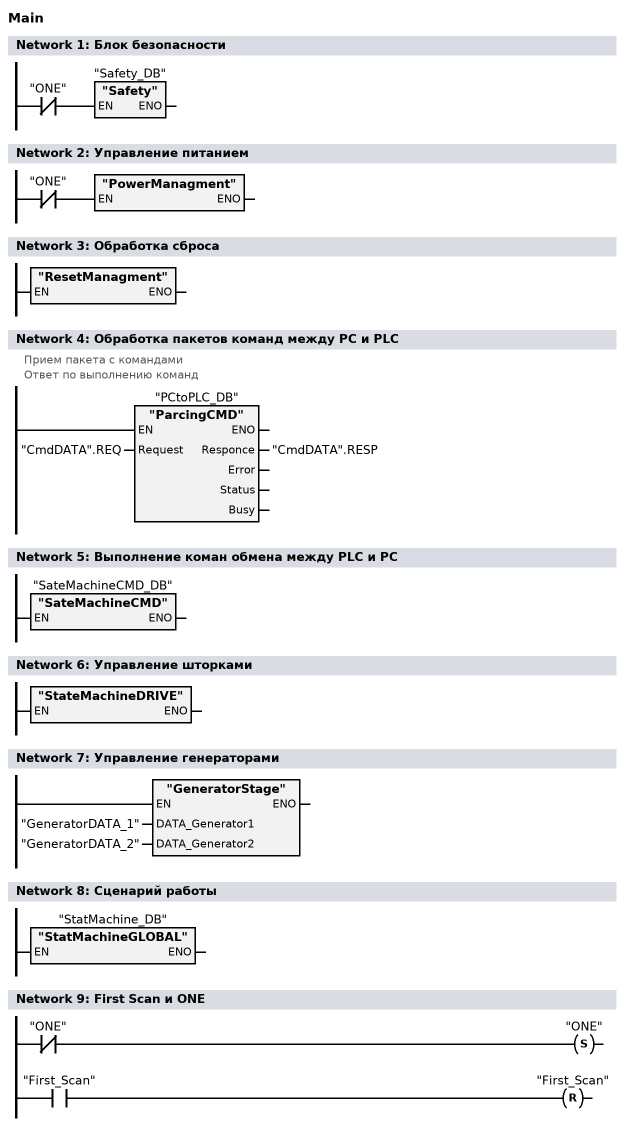
   RUNG wire#powerrail
      I_Contact( "ONE" )
      "Safety_DB"()
   END_RUNG
   // the same network as SCL:
   IF NOT "ONE" THEN
       "Safety_DB"();   // "Safety"
   END_IF;
END_REGION

REGION Network 2: Управление питанием
   RUNG wire#powerrail
      I_Contact( "ONE" )
      "PowerManagment"()
   END_RUNG
   // the same network as SCL:
   IF NOT "ONE" THEN "PowerManagment"(); END_IF;
END_REGION

REGION Network 3: Обработка сброса
   RUNG wire#powerrail
      "ResetManagment"()
   END_RUNG
   // the same network as SCL:
   "ResetManagment"();
END_REGION

REGION Network 4: Обработка пакетов команд между PC и PLC
   // Прием пакета с командами
   // Ответ по выполнению команд
   RUNG wire#powerrail
      "PCtoPLC_DB"(Request := "CmdDATA".REQ, Responce => "CmdDATA".RESP, Error =>, Status =>, Busy =>)
   END_RUNG
   // the same network as SCL:
   "PCtoPLC_DB"(Request := "CmdDATA".REQ, Responce => "CmdDATA".RESP);   // "ParcingCMD"
END_REGION

REGION Network 5: Выполнение коман обмена между PLC и PC
   RUNG wire#powerrail
      "SateMaсhineCMD_DB"()
   END_RUNG
   // the same network as SCL:
   "SateMaсhineCMD_DB"();   // "SateMaсhineCMD"
END_REGION

REGION Network 6: Управление шторками
   RUNG wire#powerrail
      "StateMachineDRIVE"()
   END_RUNG
   // the same network as SCL:
   "StateMachineDRIVE"();
END_REGION

REGION Network 7: Управление генераторами
   RUNG wire#powerrail
      "GeneratorStage"(DATA_Generator1 := "GeneratorDATA_1", DATA_Generator2 := "GeneratorDATA_2")
   END_RUNG
   // the same network as SCL:
   "GeneratorStage"(DATA_Generator1 := "GeneratorDATA_1", DATA_Generator2 := "GeneratorDATA_2");
END_REGION

REGION Network 8: Сценарий работы
   RUNG wire#powerrail
      "StatMachine_DB"()
   END_RUNG
   // the same network as SCL:
   "StatMachine_DB"();   // "StatMachineGLOBAL"
END_REGION

REGION Network 9: First Scan и ONE
   RUNG wire#powerrail
      I_Contact( "ONE" )
      S_Coil( "ONE" )
   END_RUNG
   RUNG wire#powerrail
      Contact( "First_Scan" )
      R_Coil( "First_Scan" )
   END_RUNG
   // the same network as SCL:
   IF NOT "ONE" THEN "ONE" := TRUE; END_IF;
   IF "First_Scan" THEN "First_Scan" := FALSE; END_IF;
END_REGION
END_ORGANIZATION_BLOCK

ORGANIZATION_BLOCK "Cyclic interrupt"   // OB30, LAD, CyclicInterrupt
{ S7_Optimized_Access := 'TRUE' }
VERSION : 0.1
   VAR_INPUT
      Initial_Call : Bool;   // Initial call of this OB
      Event_Count : Int;   // Events discarded
   END_VAR
BEGIN

REGION Network 1 (SCL)
       "CycleInterrupt_Flag" := TRUE;
END_REGION
END_ORGANIZATION_BLOCK

ORGANIZATION_BLOCK "Startup_1"   // OB123, LAD, Startup
TITLE = "Complete Restart"
{ S7_Optimized_Access := 'TRUE' }
VERSION : 0.1
   VAR_INPUT
      LostRetentive : Bool;   // True if retentive data are lost
      LostRTC : Bool;   // True if date and time are lost
   END_VAR
   VAR_TEMP
      i : Int;
      y : Int;
   END_VAR
   VAR CONSTANT
      T_temp : DTL;
      T_temp1 : Time;
   END_VAR
BEGIN

REGION Network 1 (SCL)
   "First_Scan" := TRUE;
   "GeneratorDATA_1".CMD_FREV := TRUE;
   "GlobalDATA".N_Presset := 1;
END_REGION

REGION Network 2 (SCL)
   "IR".Guest_index := 0;
   "IR".IR1_count := 0;
   "IR".Guest_came := 0;
   "IR".Delta_IR2_IR1 := #T_temp1;
   "IR".IR1_t1 := #T_temp;
   "IR".IR1_t2 := #T_temp;
   "IR".SHOT_make := 0;

   "KM_Generator1" := 0;

   FOR #i := 0 TO 5 BY 1
   DO
       FOR #y := 0 TO 5 BY 1
       DO
           "IR".Guest[#i].IR1[#y].t1 := #T_temp;
           "IR".Guest[#i].IR1[#y].t2 := #T_temp;
           "IR".Guest[#i].IR1[#y].delta := #T_temp1;
       END_FOR;
       "IR".Guest[#i].IR1_t1 := #T_temp;
       "IR".Guest[#i].IR2_t1 := #T_temp;
       "IR".Guest[#i].Delta_IR2_IR1 := #T_temp1;
       "IR".Guest[#i].count := 0;

   END_FOR;

   //Определяем количество снимков. Сколько генератоов будет в работе
   "GlobalDATA".Generator1.Enable := TRUE;
   "GlobalDATA".Generator2.Enable := FALSE;
   //Сервисные функции сбрасываем
   "GlobalDATA".Shutter1.cmdCycle := FALSE;
   "GlobalDATA".Shutter2.cmdCycle := FALSE;
END_REGION

REGION Network 3 (SCL): Очистка буфера обмена PC и PLC
   "GlobalDATA".REQ.ADDR := 0;
   "GlobalDATA".REQ.CMD := 0;
   "GlobalDATA".REQ.Error := FALSE;
   "GlobalDATA".REQ.Value := 0;

   "GlobalDATA".RESP.ADDR := 0;
   "GlobalDATA".RESP.CMD := 0;
   "GlobalDATA".RESP.Done := FALSE;
   "GlobalDATA".RESP.Value := 0;

   FOR #i := 0 TO 16 DO
       "CmdDATA".REQ[#i] := ' ';
       "CmdDATA".RESP[#i] := ' ';
   END_FOR;
END_REGION
END_ORGANIZATION_BLOCK

// folder: CMD

FUNCTION_BLOCK "ParcingCMD"   // FB4, SCL
{ S7_Optimized_Access := 'TRUE' }
VERSION : 0.1
   VAR_OUTPUT
      Responce : String;
      Error : Bool;   // request has error
      Status : Word;   // Status Request
      Busy : Bool;   // old comman in processing
   END_VAR
   VAR_IN_OUT
      Request : String;
   END_VAR
   VAR
      newCMD : Bool;
      ADDRBuff : Array[0..4] of Char;
      CMDBuff : Array[0..4] of Char;
      StrAddr : String;
      StrCmd : String;
      StrValue : String;
      temp_Uint : UInt;
      tempReal : Real;
      oldReq : Bool;
      ADDR : UInt;
      CMD : UInt;
      ErrorReq : Bool;
      StatusReq : Word;
      CmdCmplite : Bool;
      RespBuff : "typeRESP";
      ReqBuff : "typeREQ";
      statCountchar : UInt;
   END_VAR
   VAR_TEMP
      req : Array[0..15] of Char;
      resp : Array[0..15] of Char;
      count : UInt;
   END_VAR
BEGIN

       #newCMD := TRUE;
       #ADDR := "addrNOT";
       #CMD := "cmdNOT";
       #ErrorReq := FALSE;
       #StatusReq := "SUB_STATUS_NO_ERROR";

       REGION Read_Request_Buffer
           // Преобразование строки в массив символов
           Strg_TO_Chars(Strg := #Request,
                         pChars := 0,
                         Cnt => #count,
                         Chars := #req);

           #ReqBuff.STX := #req[0];
           #ReqBuff.ADDR[0] := #req[1];
           #ReqBuff.ADDR[1] := #req[2];
           #ReqBuff.ADDR[2] := #req[3];
           #ReqBuff.ADDR[3] := #req[4];
           #ReqBuff.hash1 := #req[5];
           #ReqBuff.CMD[0] := #req[6];
           #ReqBuff.CMD[1] := #req[7];
           #ReqBuff.CMD[2] := #req[8];
           #ReqBuff.CMD[3] := #req[9];
           #ReqBuff.hash2 := #req[10];
           #ReqBuff.VALUE[0] := #req[11];
           #ReqBuff.VALUE[1] := #req[12];
           #ReqBuff.VALUE[2] := #req[13];
           #ReqBuff.VALUE[3] := #req[14];
           #ReqBuff.CR := #req[15];
       END_REGION

       REGION STATE_PARSING    
           //Проверяем обработана ли предыдущая команда
     //      IF #oldReq = FALSE  THEN
               //Преобразуем приемный буфер адреса в строку
               //ghfhjhjy
           Chars_TO_Strg(Chars := #ReqBuff.ADDR,
                         pChars := 0,
                         Cnt := 4,
                         Strg => #StrAddr);

               //Преобразуем приемный буфер команды в строку
           Chars_TO_Strg(Chars := #ReqBuff.CMD,
                             pChars := 0,
                             Cnt := 4,
                             Strg => #StrCmd);
               // Проверка начала посылки STX=2
               IF #ReqBuff.STX <> "STX" THEN
                   #newCMD := FALSE;
               END_IF;

               //Определение адреса устройства в посылке
               IF #StrAddr = "SYSTEM" THEN
                   #ADDR := "addrSYS";
               END_IF;
               IF #StrAddr = "GENERATOR1" THEN
                   #ADDR := "addrGen1";
               END_IF;
               IF #StrAddr = "GENERATOR2" THEN
                   #ADDR := "addrGen2";
               END_IF;
               IF #StrAddr = "SHUTTER1" THEN
                   #ADDR := "addrShutter1";
               END_IF;
               IF #StrAddr = "SHUTTER2" THEN
                   #ADDR := "addrShutter2";
               END_IF;
               IF #StrAddr = "DOOR" THEN
                   #ADDR := "addrDoor";
               END_IF;
               IF #StrAddr = "DETECTOR" THEN
                   #ADDR := "addrDetector";
               END_IF;
               IF #StrAddr = "DRIVE1" THEN
                   #ADDR := "addrServoDrive1";
               END_IF;
               IF #StrAddr = "DRIVE2" THEN
                   #ADDR := "addrServoDrive2";
               END_IF;
               //Проверяем был ли вообще адрес. Если адрес не был обнаружен, то посылка не принята
               IF #ADDR = 0 THEN
                   #newCMD := FALSE;
               END_IF;

               //Проверка разделителя # Если не получен разделитель, то посылка неверная   
               IF #ReqBuff.hash1 <> "hash" THEN
                   #newCMD := FALSE;
               END_IF;

               //Определяем какая команда в посылке
               IF #StrCmd = "SETLEVEL" THEN
                   #CMD := "cmdSLEV";
               END_IF;
               IF #StrCmd = "GETLEVEL" THEN
                   #CMD := "cmdGLEV";
               END_IF;
               IF #StrCmd = "SETCURRENT" THEN
                   #CMD := "cmdSCUR";
               END_IF;
               IF #StrCmd = "GETCURRENT" THEN
                   #CMD := "cmdGCUR";
               END_IF;
               IF #StrCmd = "SETVOLTAGE" THEN
                   #CMD := "cmdSVLT";
               END_IF;
               IF #StrCmd = "GETVOLTAGE" THEN
                   #CMD := "cmdGVLT";
               END_IF;
               IF #StrCmd = "SETMODE" THEN
                   #CMD := "cmdSMOD";
               END_IF;
               IF #StrCmd = "GETMODE" THEN
                   #CMD := "cmdGMOD";
               END_IF;
               IF #StrCmd = "SETWARM" THEN
                   #CMD := "cmdSWAR";
               END_IF;
               IF #StrCmd = "GETWARM" THEN
                   #CMD := "cmdGWAR";
               END_IF;
               IF #StrCmd = "SETXRAY" THEN
                   #CMD := "cmdSRAY";
               END_IF;
               IF #StrCmd = "GETXRAY" THEN
                   #CMD := "cmdGRAY";
               END_IF;
               IF #StrCmd = "SETCLEAR" THEN
                   #CMD := "cmdSCLR";
               END_IF;
               IF #StrCmd = "GETFAULT" THEN
                   #CMD := "cmdGFLT";
               END_IF;
               IF #StrCmd = "SETPOSITION" THEN
                   #CMD := "cmdSPOS";
               END_IF;
               IF #StrCmd = "SETRESET" THEN
                   #CMD := "cmdSRES";
               END_IF;
               IF #StrCmd = "SETSCAN" THEN
                   #CMD := "cmdSCAN";
               END_IF;
               IF #StrCmd = "SETPRES1" THEN
                   #CMD := "cmdSPRESET1";
               END_IF;
               IF #StrCmd = "SETPRES2" THEN
                   #CMD := "cmdSPRESET2";
               END_IF;
               IF #StrCmd = "SETPRES3" THEN
                   #CMD := "cmdSPRESET3";
               END_IF;
               //Проверяем были ли вообще команда. Если команда не была обнаружена, то посылка не принята
               IF #CMD = 0 THEN
                   #newCMD := FALSE;
               END_IF;

               //Проверка разделителя # Если не получен разделитель, то посылка неверная   
               IF #ReqBuff.hash2 <> "hash" THEN
                   #newCMD := FALSE;
               END_IF;

               // Выделяем переданное значение
               IF #newCMD = TRUE THEN
                   Chars_TO_Strg(Chars := #ReqBuff.VALUE,
                                 pChars := 0,
                                 Cnt := 4,
                                 Strg => #StrValue);

                   STRG_VAL(IN := #StrValue,
                            FORMAT := 0,
                            P := 1,
                            OUT => #temp_Uint);

                   IF #ReqBuff.VALUE[0] < '0' OR #ReqBuff.VALUE[0] > '9' OR
                       #ReqBuff.VALUE[1] < '0' OR #ReqBuff.VALUE[1] > '9' OR
                       #ReqBuff.VALUE[2] < '0' OR #ReqBuff.VALUE[2] > '9' OR
                       #ReqBuff.VALUE[3] < '0' OR #ReqBuff.VALUE[3] > '9'
                   THEN
                       #ErrorReq := TRUE;
                       #StatusReq := "STATUS_PC_REQ_VAL_ERROR";
                   END_IF;

               END_IF;

               // Проверка окончания посылки CR=D
               IF #ReqBuff.CR <> "CR" THEN
                   #newCMD := FALSE;
               END_IF;

               //Проверка в запросе диапазона значений передаваемой величины
               //Если передаваемая велчина вне диапазона, то выставляем код ошибки
               REGION CHECK_VALUE
                   CASE #CMD OF
                       "cmdSLEV":
                           //Проверка допустимых значений Preset
                           IF #temp_Uint > 3 OR #temp_Uint < 0 THEN
                               #ErrorReq := TRUE;
                               #StatusReq := "STATUS_PC_REQ_VAL_ERROR";
                           END_IF;
                           ;
                       "cmdSCUR":
                           //Проверка допустимого значения устанавливаемого тока
                           IF #temp_Uint > "CP_max" OR #temp_Uint < "CP_min" THEN
                               #ErrorReq := TRUE;
                               #StatusReq := "STATUS_PC_REQ_VAL_ERROR";
                           END_IF;
                       "cmdSVLT":
                           //Проверка допустимого значения устанавливаемогозначения напряжения
                           #tempReal := UINT_TO_REAL(#temp_Uint);
                           #tempReal := #tempReal / 10.0;
                           IF #tempReal > "VP_max" OR #tempReal < "VP_min" THEN
                               #ErrorReq := TRUE;
                               #StatusReq := "STATUS_PC_REQ_VAL_ERROR";
                           END_IF;
                       "cmdSMOD":
                           //Проверка допустимого значения режима работы сканера
                           IF #temp_Uint > 4 THEN
                               #ErrorReq := TRUE;
                               #StatusReq := "STATUS_PC_REQ_VAL_ERROR";
                           END_IF;
                       "cmdSWAR":
                           //Проверка допустимого значения таблицы прогрева генератора
                           IF #temp_Uint > 3 THEN
                               #ErrorReq := TRUE;
                               #StatusReq := "STATUS_PC_REQ_VAL_ERROR";
                           END_IF;
                       "cmdSRAY":
                           //Проверка допустимого значения таблицы прогрева генератора
                           IF #temp_Uint > 1 THEN
                               #ErrorReq := TRUE;
                               #StatusReq := "STATUS_PC_REQ_VAL_ERROR";
                           END_IF;
                       "cmdSPOS":
                           //Проверяем номер позиции для перемещения шторки
                           IF #temp_Uint > 3 OR  #temp_Uint < 1 THEN
                               #ErrorReq := TRUE;
                               #StatusReq := "STATUS_PC_REQ_VAL_ERROR";
                           END_IF;

                       ELSE  // Statement section ELSE
                           ;
                   END_CASE;
               END_REGION  CHECK_VALUE
               // Проверяем нет ли ошибок в запросе. Если ошибок нет, то обновляем данные и выставляем флаг получения нового пакета 
               REGION NEW_CMD
                   IF #newCMD = TRUE AND #ErrorReq = FALSE THEN
                       REGION CLEAR_RESPOCE
                 //          #Responce[0] := ' ';
                 //          #Responce[1] := ' ';
                 //          #Responce[2] := ' ';
                 //          #Responce[3] := ' ';
                 //          #Responce[4] := ' ';
                 //          #Responce[5] := ' ';
                 //          #Responce[6] := ' ';
                 //          #Responce[7] := ' ';
                //           #Responce[8] := ' ';
                 //          #Responce[9] := ' ';
                //           #Responce[10] := ' ';
                //           #Responce[11] := ' ';
                 //          #Responce[12] := ' ';
                //           #Responce[13] := ' ';
                //           #Responce[14] := ' ';
                //           #Responce[15] := ' ';
                       END_REGION CLEAR_RESPONCE
                       #oldReq := TRUE;
                       "GlobalDATA".REQ.ADDR := #ADDR;
                       "GlobalDATA".REQ.CMD := #CMD;
                       "GlobalDATA".REQ.Value := #temp_Uint;

                       "GlobalDATA".RESP.ADDR := "GlobalDATA".REQ.ADDR;
                       "GlobalDATA".RESP.CMD := "GlobalDATA".REQ.CMD;


                       //Копируем номер устройства и команды из посылки запроса в поылку ответа

                       #RespBuff.ADDR[0] := #ReqBuff.ADDR[0];
                       #RespBuff.ADDR[1] := #ReqBuff.ADDR[1];
                       #RespBuff.ADDR[2] := #ReqBuff.ADDR[2];
                       #RespBuff.ADDR[3] := #ReqBuff.ADDR[3];
                       #RespBuff.CMD[0] := #ReqBuff.CMD[0];
                       #RespBuff.CMD[1] := #ReqBuff.CMD[1];
                       #RespBuff.CMD[2] := #ReqBuff.CMD[2];
                       #RespBuff.CMD[3] := #ReqBuff.CMD[3];

                   END_IF;

               //Если была ошибка в посылке, то выставляем код ошибки в запросе
               IF #newCMD = FALSE THEN
                   #ErrorReq := TRUE;
                   #StatusReq := "STATUS_PC_REQ_ERROR";
               END_IF;
           END_REGION  NEW_CMD
      //     END_IF;

       END_REGION STATE_PARSING 

       REGION STATE_RESPONCE

           IF #newCMD = TRUE OR #oldReq=TRUE THEN
               ;
               #CmdCmplite := FALSE;

               // Признак начала посылки
               #RespBuff.STX := '2';

               //Определяем к какому устройству была адресация
               REGION ADDR_CMD_VALUE
                   CASE "GlobalDATA".RESP.ADDR OF
                       "addrSYS":
                           // Выполнение системных команд
                           REGION ADRES SYSTEM                       
                               CASE "GlobalDATA".RESP.CMD OF
                                   "cmdSLEV":
                                       REGION cmdSLEV
                                           //Установка устанавливаемый номер прессета равен установленному  
                                           IF "GlobalDATA".RESP.Done= TRUE THEN
                                               "Val_to_Char"(inValue := "GlobalDATA".RESP.Value,
                                                             charBUFF => #RespBuff.VALUE);
                                               #CmdCmplite := TRUE;
                                           END_IF;
                                       END_REGION cmdSLEV
                                   "cmdGLEV":
                                       REGION cmdGLEV
                                           // Читаем установленный номер прессета
                                           "Val_to_Char"(inValue := "GlobalDATA".N_Presset,
                                                         charBUFF => #RespBuff.VALUE);
                                           #CmdCmplite := TRUE;
                                       END_REGION cmdGLEV             
                                   "cmdSMOD":
                                       REGION cmdSMOD
                                           //Устанавливаем режим работы сканера
                                           IF "GlobalDATA".modeScan = "GlobalDATA".REQ.Value THEN
                                               "Val_to_Char"(inValue := "GlobalDATA".modeScan,
                                                             charBUFF => #RespBuff.VALUE);
                                               #CmdCmplite := TRUE;
                                           END_IF;
                                       END_REGION cmdSMOD
                                   "cmdGMOD":
                                       REGION cmdGMOD
                                           //Читаем режим работы сканера
                                           "Val_to_Char"(inValue := "GlobalDATA".modeScan,
                                                         charBUFF => #RespBuff.VALUE);
                                           #CmdCmplite := TRUE;
                                       END_REGION cmdGMOD
                                   "cmdSCAN":
                                       REGION cmdSET SCAN
                                           IF "GlobalDATA".RESP.Done = TRUE THEN
                                               "Val_to_Char"(inValue := "GlobalDATA".RESP.Value,
                                                             charBUFF => #RespBuff.VALUE);
                                               #CmdCmplite := TRUE;
                                           END_IF;
                                       END_REGION cmdSET SCAN
                                   "cmdSRES":
                                       REGION cmdSET RESET GLOBAL
                                           IF "GlobalDATA".RESP.Done = TRUE THEN
                                               "Val_to_Char"(inValue := "GlobalDATA".RESP.Value,
                                                             charBUFF => #RespBuff.VALUE);
                                               #CmdCmplite := TRUE;
                                           END_IF;
                                       END_REGION cmdSET RESET GLOBAL
                                   "cmdSPRESET1" .. "cmdSPRESET3":
                                       REGION cmdSET PRESET
                                           // 
                                           IF "GlobalDATA".RESP.Done = TRUE THEN
                                               "Val_to_Char"(inValue := "GlobalDATA".RESP.Value,
                                                             charBUFF => #RespBuff.VALUE);
                                               #CmdCmplite := TRUE;
                                           END_IF;
                                       END_REGION cmdSET PRESET
                                   ELSE  // Statement section ELSE
                                       ;
                               END_CASE;
                           END_REGION ADRES_SYSTEM

                       "addrGen1":
                           // Выплнение команд генератора 1
                           REGION ADRES_GENERATOR 1
                               IF "GlobalDATA".RESP.CMD = "cmdSCUR"
                                   OR "GlobalDATA".RESP.CMD = "cmdSVLT"
                                   OR "GlobalDATA".RESP.CMD = "cmdGCUR"
                                   OR "GlobalDATA".RESP.CMD = "cmdGVLT"
                                   OR "GlobalDATA".RESP.CMD = "cmdSRAY"
                                   OR "GlobalDATA".RESP.CMD = "cmdGRAY"
                                   OR "GlobalDATA".RESP.CMD = "cmdSCLR"
                                   OR "GlobalDATA".RESP.CMD = "cmdGFLT"
                                   OR "GlobalDATA".RESP.CMD = "cmdSWAR"
                                   OR "GlobalDATA".RESP.CMD = "cmdGWAR"
                                   OR "GlobalDATA".RESP.CMD = "cmdSCAN"
                                   OR "GlobalDATA".RESP.CMD = "cmdSRES"
                               THEN
                                   // Если "GlobalDATA".RESP.Done := 1 , то команда выполнена а в "GlobalDATA".RESP.Value хранится результат
                                   IF "GlobalDATA".RESP.Done = TRUE THEN
                                       //Передаем значение после обработки команды 
                                       "Val_to_Char"(inValue := "GlobalDATA".RESP.Value,
                                                     charBUFF => #RespBuff.VALUE);
                                       #CmdCmplite := TRUE;
                                   END_IF;
                               END_IF;

                           END_REGION ADRES_GENERATOR 1

                       "addrGen2":
                           // Выплнение команд генератора 1
                           REGION ADRES_GENERATOR 2
                               IF "GlobalDATA".RESP.CMD = "cmdSCUR"
                                   OR "GlobalDATA".RESP.CMD = "cmdSVLT"
                                   OR "GlobalDATA".RESP.CMD = "cmdGCUR"
                                   OR "GlobalDATA".RESP.CMD = "cmdGVLT"
                                   OR "GlobalDATA".RESP.CMD = "cmdSRAY"
                                   OR "GlobalDATA".RESP.CMD = "cmdGRAY"
                                   OR "GlobalDATA".RESP.CMD = "cmdSCLR"
                                   OR "GlobalDATA".RESP.CMD = "cmdGFLT"
                                   OR "GlobalDATA".RESP.CMD = "cmdSWAR"
                                   OR "GlobalDATA".RESP.CMD = "cmdGWAR"
                                   OR "GlobalDATA".RESP.CMD = "cmdSRES"
                               THEN
                                   // Если "GlobalDATA".RESP.Done := 1 , то команда выполнена а в "GlobalDATA".RESP.Value хранится результат
                                   IF "GlobalDATA".RESP.Done = TRUE THEN
                                       //Передаем значение после обработки команды 
                                       "Val_to_Char"(inValue := "GlobalDATA".RESP.Value,
                                                     charBUFF => #RespBuff.VALUE);
                                       #CmdCmplite := TRUE;
                                   END_IF;
                               END_IF;

                           END_REGION ADRES_GENERATOR 2

                       "addrShutter1":
                           // Выплнение команд шторки 1
                           REGION ADRES_SHUTTER 1        
                               ;
                           END_REGION ADRES_SHUTTER 1

                       "addrShutter2":
                           // Выплнение команд шторки 2
                           REGION ADRES_SHUTTER 2    
                               ;
                           END_REGION ADRES_SHUTTER 2

                       "addrDoor":
                           // Выплнение команд двери
                           REGION DOOR    
                               IF "GlobalDATA".RESP.CMD = "cmdSRES"
                               THEN
                                   // Если "GlobalDATA".RESP.Done := 1 , то команда выполнена а в "GlobalDATA".RESP.Value хранится результат
                                   IF "GlobalDATA".RESP.Done = TRUE THEN
                                       //Передаем значение после обработки команды 
                                       "Val_to_Char"(inValue := "GlobalDATA".RESP.Value,
                                                     charBUFF => #RespBuff.VALUE);
                                       #CmdCmplite := TRUE;
                                   END_IF;
                               END_IF;
                           END_REGION DOOR

                       "addrDetector":
                           // Выплнение команд детекторов
                           REGION DETECTOR    
                               IF "GlobalDATA".RESP.CMD = "cmdSRES"
                               THEN
                                   // Если "GlobalDATA".RESP.Done := 1 , то команда выполнена а в "GlobalDATA".RESP.Value хранится результат
                                   IF "GlobalDATA".RESP.Done = TRUE THEN
                                       //Передаем значение после обработки команды 
                                       "Val_to_Char"(inValue := "GlobalDATA".RESP.Value,
                                                     charBUFF => #RespBuff.VALUE);
                                       #CmdCmplite := TRUE;
                                   END_IF;
                               END_IF;
                           END_REGION DETECTOR

                       "addrServoDrive1":
                           REGION DRIVE1    
                               IF "GlobalDATA".RESP.CMD = "cmdSPOS"
                                   OR "GlobalDATA".RESP.CMD = "cmdSRES"
                               THEN
                                   // Если "GlobalDATA".RESP.Done := 1 , то команда выполнена а в "GlobalDATA".RESP.Value хранится результат
                                   IF "GlobalDATA".RESP.Done = TRUE THEN
                                       //Передаем значение после обработки команды 
                                       "Val_to_Char"(inValue := "GlobalDATA".RESP.Value,
                                                     charBUFF => #RespBuff.VALUE);
                                       #CmdCmplite := TRUE;
                                   END_IF;
                               END_IF;
                           END_REGION DRIVE1

                       "addrServoDrive2":
                           REGION DRIVE1    
                               IF "GlobalDATA".RESP.CMD = "cmdSPOS"
                                   OR "GlobalDATA".RESP.CMD = "cmdSRES"
                               THEN
                                   // Если "GlobalDATA".RESP.Done := 1 , то команда выполнена а в "GlobalDATA".RESP.Value хранится результат
                                   IF "GlobalDATA".RESP.Done = TRUE THEN
                                       //Передаем значение после обработки команды 
                                       "Val_to_Char"(inValue := "GlobalDATA".RESP.Value,
                                                     charBUFF => #RespBuff.VALUE);
                                       #CmdCmplite := TRUE;
                                   END_IF;
                               END_IF;
                           END_REGION DRIVE1

                       ELSE  // Statement section ELSE
                           ;
                   END_CASE;

               END_REGION ADDR_CMD_VALUE

               //Признак разделителя 1
               #RespBuff.hash1 := '#';

               //Признак разделителя 2
               #RespBuff.hash2 := '#';

               //Признак окончания посылки
               #RespBuff.CR := 'D';

           END_IF;

           END_REGION STATE_RESPONCE


   REGION OUTPUT

       #Busy := #oldReq;
       #Status := #StatusReq;
       // Если в запросе передано значение VALUE вне допустимого диапазона, то возвращаем код ошибки
       IF #Status = "STATUS_PC_REQ_VAL_ERROR" THEN
           "Val_to_Char"(inValue :=  #Status,
                         charBUFF => #RespBuff.VALUE);
           #CmdCmplite := TRUE;
       END_IF;

       IF #CmdCmplite = TRUE THEN
           //Чистим приемный буфер
           #req[0] := ' ';
           #req[1] := ' ';
           #req[2] := ' ';
           #req[3] := ' ';
           #req[4] := ' ';
           #req[5] := ' ';
           #req[6] := ' ';
           #req[7] := ' ';
           #req[8] := ' ';
           #req[9] := ' ';
           #req[10] := ' ';
           #req[11] := ' ';
           #req[12] := ' ';
           #req[13] := ' ';
           #req[14] := ' ';
           #req[15] := ' ';
           Chars_TO_Strg(Chars := #req,
                         pChars := 0,
                         Cnt := 4,
                         Strg => #Request);
           // Обновляем данные в буфере обмена PLC с PC

           #resp[0] := #RespBuff.STX;
           #resp[1] := #RespBuff.ADDR[0];
           #resp[2] := #RespBuff.ADDR[1];
           #resp[3] := #RespBuff.ADDR[2];
           #resp[4] := #RespBuff.ADDR[3];
           #resp[5] := #RespBuff.hash1;
           #resp[6] := #RespBuff.CMD[0];
           #resp[7] := #RespBuff.CMD[1];
           #resp[8] := #RespBuff.CMD[2];
           #resp[9] := #RespBuff.CMD[3];
           #resp[10] := #RespBuff.hash2;
           #resp[11] := #RespBuff.VALUE[0];
           #resp[12] := #RespBuff.VALUE[1];
           #resp[13] := #RespBuff.VALUE[2];
           #resp[14] := #RespBuff.VALUE[3];
           #resp[15] := #RespBuff.CR;

           Chars_TO_Strg(Chars := #resp,
                         pChars := 0,
                         Cnt := #count,
                         Strg => #Responce);

           #Busy := FALSE;
           #oldReq := FALSE;

           "GlobalDATA".RESP.ADDR := 0;
           "GlobalDATA".RESP.CMD := 0;
           "GlobalDATA".RESP.Value := 0;

           "GlobalDATA".REQ.ADDR := 0;
           "GlobalDATA".REQ.CMD := 0;
           "GlobalDATA".REQ.Value := 0;
           "GlobalDATA".REQ.Error := 0;

           "GlobalDATA".RESP.Done := FALSE;
           #CmdCmplite := FALSE;
       END_IF;


   END_REGION OUTPUT
END_FUNCTION_BLOCK

FUNCTION_BLOCK "SateMaсhineCMD"   // FB5, SCL
{ S7_Optimized_Access := 'TRUE' }
VERSION : 0.1
   VAR
      sCP_done : Bool;
      sVP_done : Bool;
   END_VAR
   VAR_TEMP
      TempReal : Real;
      TempUint : UInt;
      err : Bool;
   END_VAR
BEGIN

   REGION STATE_MACHINE_CMD

           REGION ADDR_CMD_VALUE
               CASE "GlobalDATA".REQ.ADDR OF
                   "addrSYS":
                       // Выполнение системных команд
                       REGION ADRES SYSTEM                      
                           CASE "GlobalDATA".REQ.CMD OF
                               "cmdSLEV":
                                   REGION SETLEV
                                       //Устанавливаем номер прессета
                                       IF "GlobalDATA".REQ.Value <> "GlobalDATA".N_Presset THEN
                                           "GlobalDATA".newPreset := TRUE;
                                       END_IF;

                                       "GlobalDATA".N_Presset := "GlobalDATA".REQ.Value;

                                       //Устанавливаем значения для генератора 1
                                       "LoadPresset"(N_Presset := "GlobalDATA".N_Presset,
                  DATA_from := "PressetDATA".GUEST["GlobalDATA".N_Presset],
                  DATA_to => "GeneratorDATA_1");

                                       IF "GeneratorDATA_1".VP_Programm = "PressetDATA".GUEST["GlobalDATA".N_Presset].VP
                                           AND "GeneratorDATA_1".CP_Programm = "PressetDATA".GUEST["GlobalDATA".N_Presset].CP
                                       THEN
                                           "GeneratorDATA_1".CMD_VP := TRUE;
                                           "GeneratorDATA_1".CMD_CP := TRUE;
                                           #sCP_done := FALSE;
                                       END_IF;

                                       //Проверяем выполнение команды установки тока от генератора
                                       IF "GeneratorDATA_1".CP_Programm = "PressetDATA".GUEST["GlobalDATA".N_Presset].CP THEN
                                           IF "GeneratorDATA_1".cmdDone = TRUE AND "GeneratorDATA_1".cmd_Nunmber = "FB_STATE_CURRENT_PROGRAMM" THEN
                                               #sCP_done := TRUE;
                                           ELSIF "GeneratorDATA_1".cmdError = TRUE THEN
                                               "GlobalDATA".RESP.Value := "GeneratorDATA_1".cmdState;
                                               "GlobalDATA".RESP.Done := 1;
                                           END_IF;
                                       END_IF;
                                       //Проверяем выполнение команды установки напряжения от генератора
                                       IF "GeneratorDATA_1".VP_Programm = "PressetDATA".GUEST["GlobalDATA".N_Presset].VP THEN
                                           IF "GeneratorDATA_1".cmdDone = TRUE AND "GeneratorDATA_1".cmd_Nunmber = "FB_STATE_VOLTAGE_PROGRAMM" THEN
                                               "GlobalDATA".RESP.Done := 1;
                                               "GlobalDATA".RESP.Value := "GlobalDATA".N_Presset;
                                               "GlobalDATA".REQ.Value := 0;
                                           ELSIF "GeneratorDATA_1".cmdError = TRUE THEN
                                               "GlobalDATA".RESP.Value := "GeneratorDATA_1".cmdState;
                                               "GlobalDATA".RESP.Done := 1;
                                           END_IF;
                                       END_IF;
                                   END_REGION SETLEV
                               "cmdGLEV":
                                   REGION GETLEV
                                       //Читаем номер прессета в ответной посылке. тут сбрасываем номер команды
                                       "GlobalDATA".RESP.Done := 1;
                                       "GlobalDATA".REQ.Value := 0;
                                   END_REGION GETLEV
                               "cmdSMOD":
                                   REGION SETMOD
                                       //Устанавливаем работы сканера
                                       "GlobalDATA".modeScan := "GlobalDATA".REQ.Value;
                                       "GlobalDATA".RESP.Done := 1;
                                       "GlobalDATA".REQ.Value := 0;
                                   END_REGION SETMOD
                               "cmdGMOD":
                                   REGION GETMOD
                                       //Читаем номер прессета в ответной посылке. тут сбрасываем номер команды
                                       "GlobalDATA".RESP.Done := 1;
                                       "GlobalDATA".REQ.Value := 0;
                                   END_REGION GETMOD
                               "cmdSRES":
                                   REGION GlobalReset
                                       //Выставляем признак сброса
                                       "GlobalDATA".cmdReset.Global := TRUE;
                                       "GlobalDATA".RESP.Done := 1;
                                       "GlobalDATA".RESP.Value := "STATUS_SUBSEQUENT_CALL";
                                   END_REGION GlobalRes
                               "cmdSCAN":
                                   REGION SetScan
                                       //Выставляем признак заппуска сканирования если
                                       // есть готовность к сканированию (сканирование с X-RAY) и установлен пресет
                                       IF ("GlobalDATA".readyToScan OR NOT "GlobalDATA".Scan_XRAY) AND "GlobalDATA".N_Presset <> 0 THEN
                                           "GlobalDATA".startScan := TRUE;
                                           "GlobalDATA".RESP.Value := "STATUS_SUBSEQUENT_CALL";
                                       ELSE
                                           "GlobalDATA".RESP.Value := "ERR_UNDEFINED_STATE";
                                       END_IF;
                                       "GlobalDATA".RESP.Done := 1;

                                   END_REGION SetScan
                               "cmdSPRESET1":
                                   REGION SetSPreset1
                                       //Устанавливаем новые значения в пресета 1 если активен сервисный режим
                                       IF "GlobalDATA".modeScan = "modeSERVIСE" THEN
                                           //Выполняем рассчтеы скорости перемещения шторки и времени экспозиции для детектора исходя из требуемых значений времени экспозиции
                                           "CalcPreset"(Texposure := "GlobalDATA".REQ.Value,
                                                        Velocity => "PressetDATA".GUEST[1].Velocity,
                                                        Ttrigger => "PressetDATA".GUEST[1].Ttrigger,
                                                        Error => #err);
                                           "PressetDATA".GUEST[1].Texposure := "GlobalDATA".REQ.Value;
                                           //сли при вычислениях не боло ошибок, то возвращаем время экспозиции CareRay в мс
                                           IF #err = FALSE THEN
                                               "GlobalDATA".RESP.Value := TIME_TO_UINT("PressetDATA".GUEST[1].Ttrigger);
                                           ELSE
                                               "GlobalDATA".RESP.Value := "STATUS_PC_REQ_VAL_ERROR";
                                           END_IF;
                                       ELSE
                                          // "GlobalDATA".RESP.Value := "ERR_UNDEFINED_STATE";
                                           "GlobalDATA".RESP.Value := 200;
                                       END_IF;
                                       "GlobalDATA".RESP.Done := 1;
                                   END_REGION SetPreset1     
                               "cmdSPRESET2":
                                   REGION SetSPreset2
                                       //Устанавливаем новые значения в пресета 2 если активен сервисный режим
                                       IF "GlobalDATA".modeScan = "modeSERVIСE" THEN
                                           //Выполняем рассчтеы скорости перемещения шторки и времени экспозиции для детектора исходя из требуемых значений времени экспозиции
                                           "CalcPreset"(Texposure := "GlobalDATA".REQ.Value,
                                                        Velocity => "PressetDATA".GUEST[2].Velocity,
                                                        Ttrigger => "PressetDATA".GUEST[2].Ttrigger,
                                                        Error => #err);

                                           "PressetDATA".GUEST[2].Texposure := "GlobalDATA".REQ.Value;

                                           //сли при вычислениях не боло ошибок, то возвращаем время экспозиции CareRay в мс
                                           IF #err = FALSE THEN
                                               "GlobalDATA".RESP.Value := TIME_TO_UINT("PressetDATA".GUEST[2].Ttrigger);
                                           ELSE
                                               "GlobalDATA".RESP.Value := "STATUS_PC_REQ_VAL_ERROR";
                                           END_IF;
                                       ELSE
                                           "GlobalDATA".RESP.Value := "ERR_UNDEFINED_STATE";
                                       END_IF;
                                       "GlobalDATA".RESP.Done := 1;
                                   END_REGION SetPreset2 
                               "cmdSPRESET3":
                                   REGION SetSPreset3
                                       //Устанавливаем новые значения в пресета 1 если активен сервисный режим
                                       IF "GlobalDATA".modeScan = "modeSERVIСE" THEN
                                           //Выполняем рассчтеы скорости перемещения шторки и времени экспозиции для детектора исходя из требуемых значений времени экспозиции
                                           "CalcPreset"(Texposure := "GlobalDATA".REQ.Value,
                                                        Velocity => "PressetDATA".GUEST[3].Velocity,
                                                        Ttrigger => "PressetDATA".GUEST[3].Ttrigger,
                                                        Error => #err);
                                           "PressetDATA".GUEST[3].Texposure := "GlobalDATA".REQ.Value;
                                           //сли при вычислениях не боло ошибок, то возвращаем время экспозиции CareRay в мс
                                           IF #err = FALSE THEN
                                               "GlobalDATA".RESP.Value := TIME_TO_UINT("PressetDATA".GUEST[3].Ttrigger);
                                           ELSE
                                               "GlobalDATA".RESP.Value := "STATUS_PC_REQ_VAL_ERROR";
                                           END_IF;
                                       ELSE
                                           "GlobalDATA".RESP.Value := "ERR_UNDEFINED_STATE";
                                       END_IF;
                                       "GlobalDATA".RESP.Done := 1;
                                   END_REGION SetPreset3 
                               ELSE  // Statement section ELSE
                                   ;
                           END_CASE;
                       END_REGION ADRES_SYSTEM

                   "addrGen1":
                       // Выплнение команд генератора 1
                       REGION ADRES_GENERATOR 1
                           CASE "GlobalDATA".REQ.CMD OF
                               "cmdSCUR":
                                   REGION SET_CURRENT
                                       //Установка тока генератора
                                       IF "GeneratorDATA_1".CMD_CP = FALSE THEN
                                           "GeneratorDATA_1".CP_Programm := "GlobalDATA".REQ.Value;
                                           "GeneratorDATA_1".CMD_CP := TRUE;
                                       END_IF;
                                       //Проверяем выполнение команды от генератора
                                       IF "GeneratorDATA_1".cmdDone = TRUE AND "GeneratorDATA_1".cmd_Nunmber = "FB_STATE_CURRENT_PROGRAMM" THEN
                                           "GlobalDATA".RESP.Value := "GeneratorDATA_1".CP_Programm;
                                           "GlobalDATA".RESP.Done := 1;
                                       ELSIF "GeneratorDATA_1".cmdError = TRUE THEN
                                           "GlobalDATA".RESP.Value := "GeneratorDATA_1".cmdState;
                                           "GlobalDATA".RESP.Done := 1;
                                       END_IF;
                                   END_REGION SET_CURRENT
                               "cmdSVLT":
                                   REGION SET_VOLTAGE
                                       //Устанавливаем напряжение генератора
                                       IF "GeneratorDATA_1".CMD_VP = FALSE THEN
                                           #TempReal := UINT_TO_REAL("GlobalDATA".REQ.Value);
                                           "GeneratorDATA_1".VP_Programm := #TempReal / 10.0;
                                           "GeneratorDATA_1".CMD_VP := TRUE;
                                       END_IF;
                                       //Проверяем выполнение команды от генератора
                                       IF "GeneratorDATA_1".cmdDone = TRUE AND "GeneratorDATA_1".cmd_Nunmber = "FB_STATE_VOLTAGE_PROGRAMM" THEN
                                           #TempReal := "GeneratorDATA_1".VP_Programm * 10.0;
                                           #TempUint := REAL_TO_UINT(#TempReal);
                                           "GlobalDATA".RESP.Value := #TempUint;
                                           "GlobalDATA".RESP.Done := 1;
                                       ELSIF "GeneratorDATA_1".cmdError = TRUE THEN
                                           "GlobalDATA".RESP.Value := "GeneratorDATA_1".cmdState;
                                           "GlobalDATA".RESP.Done := 1;
                                       END_IF;
                                   END_REGION SET_VOLTAGE
                               "cmdGCUR":
                                   REGION GET_CURRENT
                                       //Чтение тока генератора
                                       "GeneratorDATA_1".CMD_MON := TRUE;

                                       //Проверяем выполнение команды от генератора
                                       IF "GeneratorDATA_1".cmdDone = TRUE AND "GeneratorDATA_1".cmd_Nunmber = "FB_STATE_MONITOR" THEN
                                           "GlobalDATA".RESP.Value := "GeneratorDATA_1".CP_Monitor;
                                           "GlobalDATA".RESP.Done := 1;
                                       ELSIF "GeneratorDATA_1".cmdError = TRUE THEN
                                           "GlobalDATA".RESP.Value := "GeneratorDATA_1".cmdState;
                                           "GlobalDATA".RESP.Done := 1;
                                       END_IF;
                                   END_REGION GET_CURRENT
                               "cmdGVLT":
                                   REGION GET_VALUE
                                       //Чтение напряжения генератора
                                       "GeneratorDATA_1".CMD_MON := TRUE;

                                       //Проверяем выполнение команды от генератора
                                       IF "GeneratorDATA_1".cmdDone = TRUE AND "GeneratorDATA_1".cmd_Nunmber = "FB_STATE_MONITOR" THEN
                                           #TempReal := "GeneratorDATA_1".VP_Monitor * 10.0;
                                           #TempUint := REAL_TO_UINT(#TempReal);
                                           "GlobalDATA".RESP.Value := #TempUint;
                                           "GlobalDATA".RESP.Done := 1;
                                       ELSIF "GeneratorDATA_1".cmdError = TRUE THEN
                                           "GlobalDATA".RESP.Value := "GeneratorDATA_1".cmdState;
                                           "GlobalDATA".RESP.Done := 1;
                                       END_IF;
                                   END_REGION GET_VALUE
                               "cmdSRAY":
                                   REGION SET_XRAY
                                       //Включение X-RAY если шторка находится в закрытом положении
                                       IF "GlobalDATA".Shutter1.setPOS1 OR "GlobalDATA".Shutter1.setPOS2 THEN
                                           IF "GlobalDATA".REQ.Value = 1 THEN
                                               "GlobalDATA"."Generator1".CmdXRAY_ON := TRUE;
                                           ELSIF "GlobalDATA".REQ.Value = 0 THEN
                                               "GlobalDATA"."Generator1".CmdXRAY_ON := FALSE;
                                           END_IF;

                                           //Проверяем статус генератора
                                           IF "GeneratorDATA_1".cmdDone = TRUE AND "GeneratorDATA_1".cmd_Nunmber = "FB_STATE_MONITOR" THEN
                                               IF ("GlobalDATA".REQ.Value = 1 AND "GlobalDATA".Generator1.XRAY_Status = TRUE) THEN
                                                   "GlobalDATA".RESP.Value := 1;
                                                   "GlobalDATA".RESP.Done := 1;
                                               END_IF;
                                               IF ("GlobalDATA".REQ.Value = 0 AND "GlobalDATA".Generator1.XRAY_Status = FALSE) THEN
                                                   "GlobalDATA".RESP.Value := 0;
                                                   "GlobalDATA".RESP.Done := 1;
                                               END_IF;
                                               IF "GeneratorDATA_1".cmdError = TRUE THEN
                                                   "GlobalDATA".RESP.Value := "GeneratorDATA_1".cmdState;
                                                   "GlobalDATA".RESP.Done := 1;
                                               END_IF;
                                           END_IF;
                                       ELSE
                                           "GlobalDATA".RESP.Value := "ERR_UNDEFINED_STATE";
                                           "GlobalDATA".RESP.Done := 1;
                                       END_IF;
                                   END_REGION SET_XRAY
                               "cmdGRAY":
                                   REGION GET_XRAY_STATUS
                                       //Проверяем статус генератора
                                       "GeneratorDATA_1".CMD_STAT := TRUE;
                                       IF "GeneratorDATA_1".cmdDone = TRUE AND "GeneratorDATA_1".cmd_Nunmber = "FB_STATE_HV_STATUS" THEN
                                           IF "GeneratorDATA_1".X_RAY_Status = TRUE THEN
                                               "GlobalDATA".RESP.Value := 1;
                                           ELSE
                                               "GlobalDATA".RESP.Value := 0;
                                           END_IF;
                                           "GlobalDATA".RESP.Done := 1;
                                       ELSIF "GeneratorDATA_1".cmdError = TRUE THEN
                                           "GlobalDATA".RESP.Value := "GeneratorDATA_1".cmdState;
                                           "GlobalDATA".REQ.CMD := 0;
                                       END_IF;
                                   END_REGION GET_XRAY_STATUS
                               "cmdSWAR":
                                   REGION SET_WARM
                                       //Установка режима прогрева генератора
                                       IF "GlobalDATA".Generator1.Ready = TRUE THEN
                                           "GlobalDATA".Generator1.cmdWarm := "GlobalDATA".REQ.Value;
                                           IF "GlobalDATA".Generator1.warmEN THEN
                                               "GlobalDATA".RESP.Done := 1;
                                               //Возвращаем код выполнения программы без ошибок
                                               "GlobalDATA".RESP.Value := "GlobalDATA".Generator1.cmdWarm;;
                                           END_IF;
                                       ELSE
                                           //Если генератор был не готов, то выдаем ошибку
                                           "GlobalDATA".RESP.Done := 1;
                                           "GlobalDATA".RESP.Value := "ERR_UNDEFINED_STATE";
                                       END_IF;
                                   END_REGION SET_WARM
                               "cmdGWAR":
                                   REGION GET_WARM
                                       //Если генератор готов и идет прогрев, то возвращаем значение таблицы прогрева
                                       IF "GlobalDATA".Generator1.Ready = TRUE AND "GlobalDATA".Generator1.warmEN THEN
                                           //Возвращаем код выполнения программы без ошибок
                                           "GlobalDATA".RESP.Value := "GlobalDATA".Generator1.cmdWarm;
                                       ELSE
                                           //Если генератор был не готов или не выполняется прогрев, то выдаем ошибку
                                           "GlobalDATA".RESP.Value := "STATUS_NO_CALL";
                                       END_IF;
                                       "GlobalDATA".RESP.Done := 1;
                                   END_REGION GET_WARM
                               "cmdSCLR":
                                   REGION SET_CLEAR_FAULT
                                       //Сброс ошибок генератора
                                       "GeneratorDATA_1".CMD_CLR := TRUE;
                                       //Проверяем выполнение команды от генератора
                                       IF "GeneratorDATA_1".cmdDone = TRUE AND "GeneratorDATA_1".cmd_Nunmber = "FB_STATE_FAULT_CLEAR" THEN
                                           //Чтение ошибок генератора
                                           "GeneratorDATA_1".CMD_FLT := TRUE;
                                       END_IF;

                                       //Проверяем выполнение команды от генератора
                                       IF "GeneratorDATA_1".cmdDone = TRUE AND "GeneratorDATA_1".cmd_Nunmber = "FB_STATE_REPORT_FAULT" THEN
                                           "GlobalDATA".RESP.Value.%X0 := "GeneratorDATA_1".FLT[0];
                                           "GlobalDATA".RESP.Value.%X1 := "GeneratorDATA_1".FLT[1];
                                           "GlobalDATA".RESP.Value.%X2 := "GeneratorDATA_1".FLT[2];
                                           "GlobalDATA".RESP.Value.%X3 := "GeneratorDATA_1".FLT[3];
                                           "GlobalDATA".RESP.Value.%X4 := "GeneratorDATA_1".FLT[4];
                                           "GlobalDATA".RESP.Value.%X5 := "GeneratorDATA_1".FLT[5];
                                           "GlobalDATA".RESP.Value.%X6 := "GeneratorDATA_1".FLT[6];
                                           "GlobalDATA".RESP.Value.%X7 := "GeneratorDATA_1".FLT[7];
                                           "GlobalDATA".RESP.Value.%X8 := "GeneratorDATA_1".FLT[8];
                                           "GlobalDATA".RESP.Done := 1;
                                       ELSIF "GeneratorDATA_1".cmdError = TRUE THEN
                                           "GlobalDATA".RESP.Value := "GeneratorDATA_1".cmdState;
                                           "GlobalDATA".RESP.Done := 1;
                                       END_IF;
                                   END_REGION SET_CLEAR_FAULT
                               "cmdGFLT":
                                   REGION GET_FAULT
                                       //Чтение ошибок генератора
                                       "GeneratorDATA_1".CMD_FLT := TRUE;

                                       //Проверяем выполнение команды от генератора
                                       IF "GeneratorDATA_1".cmdDone = TRUE AND "GeneratorDATA_1".cmd_Nunmber = "FB_STATE_REPORT_FAULT" THEN
                                           "GlobalDATA".RESP.Value.%X0 := "GeneratorDATA_1".FLT[0];
                                           "GlobalDATA".RESP.Value.%X1 := "GeneratorDATA_1".FLT[1];
                                           "GlobalDATA".RESP.Value.%X2 := "GeneratorDATA_1".FLT[2];
                                           "GlobalDATA".RESP.Value.%X3 := "GeneratorDATA_1".FLT[3];
                                           "GlobalDATA".RESP.Value.%X4 := "GeneratorDATA_1".FLT[4];
                                           "GlobalDATA".RESP.Value.%X5 := "GeneratorDATA_1".FLT[5];
                                           "GlobalDATA".RESP.Value.%X6 := "GeneratorDATA_1".FLT[6];
                                           "GlobalDATA".RESP.Value.%X7 := "GeneratorDATA_1".FLT[7];
                                           "GlobalDATA".RESP.Value.%X8 := "GeneratorDATA_1".FLT[8];
                                           "GlobalDATA".RESP.Done := 1;
                                       ELSIF "GeneratorDATA_1".cmdError = TRUE THEN
                                           "GlobalDATA".RESP.Value := "GeneratorDATA_1".cmdState;
                                           "GlobalDATA".RESP.Done := 1;
                                       END_IF;
                                   END_REGION GET_FAULT
                               "cmdSRES":
                                   REGION SET_RESET
                                       //Выставляем признак сброса
                                       "GlobalDATA".cmdReset.Generator1 := TRUE;
                                       "GlobalDATA".RESP.Done := 1;
                                       "GlobalDATA".RESP.Value := "STATUS_SUBSEQUENT_CALL";
                                   END_REGION SET_RESET
                           END_CASE;
                       END_REGION ADRES_GENERATOR 1

